(* IEC 61131-3 sources: BLM_BACKGROUND/src/PROGRAM_FILES/FB (part 3) *)

        _FB_Jog_Asse#STATE_JOG_ASSE_POS_ASSE_POSITIVE:
              IF (PosAsse.outputState<>GENERAL_STATE#STATE_END) THEN
                  PosAsse(AttesaResetAxes:=TRUE,
                                  axis:=Axes[Asse].PosAx,
                                  //direction:=BY_VALUE,
                                  //positioningMode:=pMode,
                                  position:=corsa,
                                  //velocityType:=DIRECT,
                                  velocity:=jogvel,
                                  //positiveAccelType:=DIRECT,
                                  //negativeAccelType:=DIRECT,
                                  positiveAccel:=jogacc,
                                  negativeAccel:=jogacc
                                  //velocityProfile:=TRAPEZOIDAL,
                                  //blendingMode:=INACTIVE,
                                  //mergeMode:=IMMEDIATELY,
                                  //nextCommand:=IMMEDIATELY
                                  );
              ELSE
                  PosAsse(AttesaResetAxes:=TRUE,
                                  axis:=Axes[Asse].PosAx,
                                  //direction:=BY_VALUE,
                                  //positioningMode:=pMode,
                                  position:=corsa,
                                  //velocityType:=DIRECT,
                                  velocity:=jogvel,
                                  //positiveAccelType:=DIRECT,
                                  //negativeAccelType:=DIRECT,
                                  positiveAccel:=jogacc,
                                  negativeAccel:=jogacc
                                  //velocityProfile:=TRAPEZOIDAL,
                                  //blendingMode:=INACTIVE,
                                  //mergeMode:=IMMEDIATELY,
                                  //nextCommand:=IMMEDIATELY
                                  );
                  CURRENT_STATE:=_FB_Jog_Asse#STATE_JOG_ASSE_JOG_PURO_NEGATIVO;
              END_IF;

        _FB_Jog_Asse#STATE_JOG_ASSE_JOG_PURO_NEGATIVO:
            //   {::ifdef BLOCCAGGIO_DX} %%%%% non c'e in config di machina
            //       IF Asse=W3 THEN
            //           AppoDirezione:=SN;
            //       ELSE
            //           AppoDirezione:=SN_SP;
            //       END_IF;
            //   {::else}
            //       AppoDirezione:=SN_SP;
            //   {::endif}
              IF ((r_minus.Q=TRUE) AND (Clk_plus=FALSE)) OR
                   ((Clk_plus=FALSE) AND (Clk_minus=TRUE) AND (r_rapid.Q=TRUE)) OR
                   ((Clk_minus=TRUE) AND (Clk_plus=FALSE) AND (f_rapid.q=TRUE)) THEN
                  IF OK_Condizione_Move_Asse(Asse:=Asse, Direzione:=AppoDirezione) THEN
                      reset_trace(Code:=TRC_SAFETY_JOG_DEVICES);
                      IF i_sys_varinc=0 THEN
                          // è in JOG puro e non incrementale
                          //limite negativo attivo
                          PosAx:= AsSynchronousAxisRef(Axes[asse].PosAx);
                          corsa:=PosAx^.PositionLimits_SW.MinPosition+EXTRALIMIT;
                          //corsa:=Axes[asse].PosAx.swlimit.minusposition+EXTRALIMIT;
                          pMode:=_EnumPositioningMode#ABSOLUTE;
                      ELSE
                          IF i_sys_varinc>=1 AND i_sys_varinc<=5 THEN
                              // valore fisso
                              corsa:=-INC[i_sys_varinc];

                              corsa:=INC_Enum#inc_0;
                              pMode:=_EnumPositioningMode#RELATIVE;
                            //   Axes[Asse].mcJogAxisInfo.Increment:=corsa; //???????
                            //   Axes[Asse].mcJogAxisInfo.ModeInc:=TRUE;
                          ELSE  // Quota target
                              //Se la quota supera il fine corsa la limita
                              PosAx:= AsSynchronousAxisRef(Axes[asse].PosAx);
                                IF pm[asse].MA_JOG_TARGET<PosAx^.PositionLimits_SW.MinPosition THEN
                                pm[asse].MA_JOG_TARGET:=PosAx^.PositionLimits_SW.MinPosition+EXTRALIMIT;
                              //IF pm[asse].MA_JOG_TARGET<Axes[asse].PosAx.swlimit.minusposition THEN
                                  //pm[asse].MA_JOG_TARGET:=Axes[asse].PosAx.swlimit.minusposition+EXTRALIMIT;
                              END_IF;
                              // se l^asse è oltre la quota target
                              PosAx:= AsSynchronousAxisRef(Axes[asse].PosAx);
                            //   IF Posax^.actualposition-Axes[Asse].Posax.servosettings.additionalcommandvalue[0]-0.1<pm[asse].MA_JOG_TARGET THEN ???
                            //       corsa:=PosAx^.PositionLimits_SW.MinPosition +EXTRALIMIT;
                            //   ELSE
                            //       // valore fisso
                            //       corsa:=pm[asse].MA_JOG_TARGET;
                            //   END_IF;
                              pMode:=_EnumPositioningMode#ABSOLUTE;
                          END_IF;
                      END_IF;
                  END_IF;
                  IF i_sys_monitoring<>0 OR i_sys_Accesslevel<=ACCESS_MANUTENTORE OR SbloccaMonitoring(Asse:=Asse)=TRUE THEN
                      IF Sbloccamonitoring(Asse:=Asse)=TRUE OR i_sys_monitoring=0 THEN
                          set_trace(Code:=TRC_MONITORING_DISABILITATO);
                      END_IF;// muove solo se in monitoring o con livello password alto e non è oltre il finecorsa negativo
                      PosAx:= AsSynchronousAxisRef(Axes[asse].PosAx);
                      IF Posax^.actualposition-0.01>PosAx^.PositionLimits_SW.MinPosition+EXTRALIMIT THEN
                          TestAsseUtensile(Asse);
                          i_sys_PosFinale[Asse]:=corsa;
                          IF (pMode=_EnumPositioningMode#RELATIVE AND USOPLCOpen) THEN
                              //Axes[Asse].mcJogAxisInfo.Enable:=TRUE;
                              Axes[Asse].MC_Axes.move_jog_param.JogBackward :=TRUE;
                              //Axes[Asse].mcJogAxisInfo.Backward:=TRUE;
                          ELSE
                              CURRENT_STATE:=_FB_Jog_Asse#STATE_JOG_ASSE_POS_ASSE_NEGATIVE;
                          END_IF;
                      ELSE
                          CURRENT_STATE:=_FB_Jog_Asse#STATE_JOG_ASSE_RILASCIO_PULSANTI;
                      END_IF;
                  ELSE
                      set_trace(Code:=TRC_JOG_NON_IN_MONITORING);
                      CURRENT_STATE:=_FB_Jog_Asse#STATE_JOG_ASSE_RILASCIO_PULSANTI;
                  END_IF;
              ELSE
                  CURRENT_STATE:=_FB_Jog_Asse#STATE_JOG_ASSE_RILASCIO_PULSANTI;
              END_IF;

        _FB_Jog_Asse#STATE_JOG_ASSE_POS_ASSE_NEGATIVE:
              IF (PosAsse.outputState<>GENERAL_STATE#STATE_END) THEN
                  PosAsse(AttesaResetAxes:=TRUE,
                                  axis:=Axes[Asse].PosAx,
                                  //direction:=BY_VALUE,
                                  positioningMode:=pMode,
                                  position:=corsa,
                                  //velocityType:=DIRECT,
                                  velocity:=jogvel,
                                  //positiveAccelType:=DIRECT,
                                  //negativeAccelType:=DIRECT,
                                  positiveAccel:=jogacc,
                                  negativeAccel:=jogacc
                                  //velocityProfile:=TRAPEZOIDAL,
                                  //blendingMode:=INACTIVE,
                                  //mergeMode:=IMMEDIATELY,
                                  //nextCommand:=IMMEDIATELY
                                  );
              ELSE
                  PosAsse(AttesaResetAxes:=TRUE,
                                  axis:=Axes[Asse].PosAx,
                                  //direction:=BY_VALUE,
                                  positioningMode:=pMode,
                                  position:=corsa,
                                  //velocityType:=DIRECT,
                                  velocity:=jogvel,
                                  //positiveAccelType:=DIRECT,
                                  //negativeAccelType:=DIRECT,
                                  positiveAccel:=jogacc,
                                  negativeAccel:=jogacc
                                  //velocityProfile:=TRAPEZOIDAL,
                                  //blendingMode:=INACTIVE,
                                  //mergeMode:=IMMEDIATELY,
                                  //nextCommand:=IMMEDIATELY
                                  );
                  CURRENT_STATE:=_FB_Jog_Asse#STATE_JOG_ASSE_RILASCIO_PULSANTI;
              END_IF;

        _FB_Jog_Asse#STATE_JOG_ASSE_RILASCIO_PULSANTI:
              //RILASCIATO TASTO ^+^ oppure RILASCIATO TASTO ^-^
              IF (f_plus.q=TRUE) OR (f_minus.q=TRUE) OR
                   ((r_plus.q=TRUE) AND (Clk_minus=TRUE)) OR
                   ((r_minus.q=TRUE) AND (Clk_plus=TRUE)) THEN
                  i_sys_posfinale[asse]:=-MY_BIG_VALUE_REAL;
                  IF (Axes[Asse].MC_Axes.State_move_jog.Busy) THEN
                    Axes[Asse].MC_Axes.move_jog_param.JogBackward :=FALSE;
                    Axes[Asse].MC_Axes.move_jog_param.JogForward :=FALSE;
                    //   Axes[Asse].mcJogAxisInfo.Backward:=FALSE;
                    //   Axes[Asse].mcJogAxisInfo.Forward:=FALSE;
                      //Axes[Asse].mcJogAxisInfo.Enable:=FALSE;
                  ELSE
                      StopAxis(asse:=asse  , Acceleration:=jogacc (*Deceleration:=jogacc*));
                  END_IF;
                  reset_trace(TRC_JOG_NON_IN_MONITORING);
                  reset_trace(Code:=TRC_MONITORING_DISABILITATO);
                  CURRENT_STATE:=GENERAL_STATE#STATE_END;
              ELSE
                  CURRENT_STATE:=GENERAL_STATE#STATE_END;
              END_IF;

          GENERAL_STATE#STATE_END:
              CURRENT_STATE:=GENERAL_STATE#STATE_INIT;

      END_CASE;
      OutputState:=CURRENT_STATE;
  END_FUNCTION_BLOCK

  FUNCTION_BLOCK FB_MuoviDispositivo

    VAR_EXTERNAL CONSTANT
        FIRST_DEVICE                          :INT;
    END_VAR

    VAR_INPUT
      Dispositivo    :INT;
      Stato          :INT;
    END_VAR
    VAR
      Esito            :BOOL;
      AppoStato        :INT;
      dret         		 :DINT;

          CURRENT_STATE				:INT:=GENERAL_STATE#STATE_INIT;
        //   {#ifndef ORBITALE}
        //       PinzaCoccodrillo	:FB_PinzaCoccodrillo;
        //   {#endif};
    END_VAR
      VAR_OUTPUT
          OutputState					:INT;
      END_VAR
      CASE CURRENT_STATE OF
          GENERAL_STATE#STATE_INIT:
              IF Dispositivo>=FIRST_DEVICE AND Dispositivo<=FIRST_DEVICE+_MAXDEVICES#MAXDEVICES-1 THEN
                //   {#ifdef ORBITALE}
                //       IF Disp[Dispositivo].TipoOut=DISP_OUT_V_C THEN
                //           AppoStato:=Stato;
                //           {#ifdef DH4010}
                //               IF Dispositivo=PINZA_SX OR Dispositivo=PINZA_DX THEN
                //                   //Gestione chiusura pinza su 2 posizioni. Se si parte da INTERMEDIO si può attivare LAVORO,
                //                   //altrimenti si attiva INTERMEDIO
                //                   IF Stato=LAVORO OR Stato=INTERMEDIO_PINZA THEN
                //                       IF Disp[Dispositivo].stato=INTERMEDIO_PINZA THEN
                //                           AppoStato:=LAVORO;
                //                       ELSE
                //                           AppoStato:=INTERMEDIO_PINZA;
                //                       END_IF;
                //                   END_IF;
                //                   IF Stato=RIPOSO OR Stato=INTERMEDIO_PINZA THEN
                //                       IF Disp[Dispositivo].stato=INTERMEDIO_PINZA THEN
                //                           AppoStato:=RIPOSO;
                //                       ELSE
                //                           AppoStato:=INTERMEDIO_PINZA;
                //                       END_IF;
                //                   END_IF;
                //               END_IF;
                //           {#endif}	//Fine DH4010
                //           Set_Disp_Position(Ndisp:=Dispositivo, Value:=AppoStato, TimerRisparmio:=TRUE);
                //           CURRENT_STATE:=GENERAL_STATE#STATE_END;
                //       ELSE
                //           set_disp(Ndisp:=Dispositivo, Stato:=Stato, TimerRisparmio:=TRUE);
                //           CURRENT_STATE:=GENERAL_STATE#STATE_END;
                //       END_IF;
                //   {#else}  //Fine ORBITALE
                //       IF Dispositivo=PINZA THEN
                //           IF cfg.UsoPinzaCoccoPneumatica=TRUE AND programmi[PROGRAMMA_JOG].PinzaCoccodrillo3Posizioni=TRUE THEN
                //               IF Stato=RIPOSO AND  Disp[PINZA].position=LAVORO THEN
                //                   AppoStato:=PREAPERTO;
                //               ELSE
                //                   AppoStato:=Stato;
                //               END_IF;
                //               CURRENT_STATE:=STATE_MUOVI_DISPOSITIVO_PINZA_COCCODRILLO;
                //           ELSE
                //               WriteDigitalOutput(NumOutput:=OUT_PREAPERTURA_PINZA_COCCODRILLO, Value:=FALSE);
                //               WriteDigitalOutput(NumOutput:=OUT_RESET_PINZA_COCCODRILLO_PREAPERTA, Value:=TRUE);
                //               set_disp(Ndisp:=Dispositivo, Stato:=Stato, TimerRisparmio:=TRUE);
                //               CURRENT_STATE:=GENERAL_STATE#STATE_END;
                //           END_IF;
                //       ELSE
                //           set_disp(Ndisp:=Dispositivo, Stato:=Stato, TimerRisparmio:=TRUE);
                //           CURRENT_STATE:=GENERAL_STATE#STATE_END;
                //       END_IF;
                //   {#endif}  //Fine NO ORBITALE
            //   ELSE
                  CURRENT_STATE:=GENERAL_STATE#STATE_END;
              END_IF;

        //   STATE_MUOVI_DISPOSITIVO_PINZA_COCCODRILLO:
        //   ;
            //   {#ifndef ORBITALE} %%%%
            //       IF PinzaCoccodrillo.OutputState<>GENERAL_STATE#STATE_END THEN
            //           PinzaCoccodrillo(Stato:=AppoStato,
            //                                            FlagStopPoint:=FALSE,
            //                                            Impostazione:=TRUE,
            //                                            Attesa:=FALSE,
            //                                            Trace:=FALSE);
            //       ELSE
            //           Esito:=PinzaCoccodrillo.ReturnValue;
            //           PinzaCoccodrillo();
            //           Disp[PINZA].position:=AppoStato;
            //           Disp[PINZA].stato:=AppoStato;
            //           CURRENT_STATE:=GENERAL_STATE#STATE_END;
            //       END_IF;
            //   {#endif};

          GENERAL_STATE#STATE_END:
              CURRENT_STATE:=GENERAL_STATE#STATE_INIT;

      END_CASE;
      OutputState:=CURRENT_STATE;
  END_FUNCTION_BLOCK

  FUNCTION_BLOCK FB_PosizionaSostegno
    VAR_INPUT
      Posizione :LREAL;
      Attesa    :BOOL:=TRUE;
    END_VAR
    VAR
      dret      :DINT;
      PosS1     :LREAL;
      OffsetS1  :LREAL;
      Programma :DINT;

          CURRENT_STATE				:INT:=GENERAL_STATE#STATE_INIT;
        //   Wait_Disp_Position	:FB_Wait_Disp_Position; %%%%
        //   PosAxeNoWait				:FB_PosAxeNoWait;
        //   WaitAxe							:FB_WaitAxe;
          EnableAxisBLM				:FB_EnableAxisBLM;
    END_VAR
      VAR_OUTPUT
          OutputState					:INT;
      END_VAR
      ;
    //   CASE CURRENT_STATE OF %%%%
    //       GENERAL_STATE#STATE_INIT:
    //           {#ifndef ORBITALE}
    //               {#ifdef SOSTEGNO_ELETTRICO}
    //                   //Impostazione dell^indice del pezzo attivo, se non siamo in AUTO il pezzo
    //                   //attivo da dove prendere i dati è 1
    //                   IF i_sys_OPMODE=AUTOMODE THEN
    //                       Programma:=i_sys_current_prog;
    //                   ELSE
    //                       Programma:=PROGRAMMA_JOG;
    //                   END_IF;
    //                   IF Assi[S1].PosAx.positioningState.homed=YES AND pm[S1].ma_stato_index=2 THEN
    //                       IF Programmi[Programma].diametro_tubo_sezione=TONDO THEN
    //                           //Gestione tubo tondo, la posizione S1 è calcolata direttamente da VGP
    //                           OffsetS1:=BlmMxToolsOffPezzo[(S1)].PosChiuso-
    //                                               BlmMxToolsOffPezzo[(S1)].Offset;
    //                           IF ABS(Posizione-RIPOSO)<=pm[S1].ma_tolerance OR
    //                                ABS(Posizione-BlmMxToolsOffPezzo[(S1)].PosAperto)<=pm[S1].ma_tolerance THEN
    //                               //Posizione bassa sostegno non si applica l^offset
    //                               PosS1:=BlmMxToolsOffPezzo[(S1)].PosAperto;
    //                           ELSE
    //                               IF ABS(Posizione-LAVORO)<=pm[S1].ma_tolerance THEN
    //                                   PosS1:=BlmMxToolsOffPezzo[(S1)].offset;
    //                               ELSE
    //                                   PosS1:=Posizione-OffsetS1;
    //                               END_IF;
    //                           END_IF;
    //                       ELSE
    //                           //Tubi non tondi la posizione di S1 dipende dalla posizione di Z1
    //                           IF ABS(Posizione-RIPOSO)<=pm[S1].ma_tolerance OR
    //                                ABS(Posizione-BlmMxToolsOffPezzo[(S1)].PosAperto)<=pm[S1].ma_tolerance THEN
    //                               //Posizione bassa sostegno non si applica l^offset
    //                               PosS1:=BlmMxToolsOffPezzo[(S1)].PosAperto;
    //                           ELSE
    //                               //Richiesta posizione alta occorre calcolarla in funzione di Z1
    //                               PosS1:=CalcS1daZ1(PosZ1:=Assi[Z1].PosAx.positioningState.actualPosition+
    //                                                                                Programmi[Programma].OffsetZ1RicSaldatura,
    //                                                                   Programma:=Programma,
    //                                                                   Sezione:=Programmi[Programma].diametro_tubo_sezione);
    //                           END_IF;
    //                       END_IF;
    //                       IF Attesa=FALSE AND Assi[S1].PosAx.control<>ACTIVE  THEN
    //                           CURRENT_STATE:=STATE_POSIZIONA_SOSTEGNO_ENABLE_SOSTEGNO;
    //                       ELSE
    //                           CURRENT_STATE:=STATE_POSIZIONA_SOSTEGNO_POS_SOSTEGNO_ELETTRICO;
    //                       END_IF;
    //                   ELSE
    //                       CURRENT_STATE:=GENERAL_STATE#STATE_END;
    //                   END_IF;
    //               {#else}
    //                   Set_disp_Position(Ndisp:=SUPPORT_TIRANT, Value:=Posizione, TimerRisparmio:=TRUE);
    //                   IF Attesa=TRUE THEN
    //                       CURRENT_STATE:=STATE_POSIZIONA_SOSTEGNO_WAIT_SOSTEGNO_PNEUMATICO;
    //                   ELSE
    //                       CURRENT_STATE:=GENERAL_STATE#STATE_END;
    //                   END_IF;
    //               {#endif}
    //           {#else}
    //               CURRENT_STATE:=GENERAL_STATE#STATE_END;
    //           {#endif};

    //       STATE_POSIZIONA_SOSTEGNO_POS_SOSTEGNO_ELETTRICO:
    //           {#ifdef SOSTEGNO_ELETTRICO}
    //               IF (PosAxeNoWait.outputState<>GENERAL_STATE#STATE_END) THEN
    //                   PosAxeNoWait(Quota:=PosS1, Asse:=S1);
    //               ELSE
    //                   PosAxeNoWait(Quota:=PosS1, Asse:=S1);
    //                   IF Attesa THEN
    //                       CURRENT_STATE:=STATE_POSIZIONA_SOSTEGNO_WAIT_SOSTEGNO_ELETTRICO;
    //                   ELSE
    //                       CURRENT_STATE:=GENERAL_STATE#STATE_END;
    //                   END_IF;
    //               END_IF;
    //           {#endif};

    //       STATE_POSIZIONA_SOSTEGNO_WAIT_SOSTEGNO_ELETTRICO:
    //           {#ifdef SOSTEGNO_ELETTRICO}
    //               IF (WaitAxe.outputState<>GENERAL_STATE#STATE_END) THEN
    //                   WaitAxe(Quota:=PosS1, Asse:=S1);
    //               ELSE
    //                   WaitAxe(Quota:=PosS1, Asse:=S1);
    //                   CURRENT_STATE:=GENERAL_STATE#STATE_END;
    //               END_IF;
    //           {#endif};

    //       STATE_POSIZIONA_SOSTEGNO_ENABLE_SOSTEGNO:
    //           {#ifdef SOSTEGNO_ELETTRICO}
    //               IF (EnableAxisBLM.outputState<>GENERAL_STATE#STATE_END) THEN
    //                   EnableAxisBLM(Asse:=assi[S1].PosAx,
    //                                               NumeroAsse:=S1,
    //                                               ModoAttesa:=IMMEDIATELY);
    //               ELSE
    //                   EnableAxisBLM(Asse:=assi[S1].PosAx,
    //                                               NumeroAsse:=S1,
    //                                               ModoAttesa:=IMMEDIATELY);
    //                   CURRENT_STATE:=GENERAL_STATE#STATE_END;
    //               END_IF;
    //           {#endif};

    //       STATE_POSIZIONA_SOSTEGNO_WAIT_SOSTEGNO_PNEUMATICO:
    //           {#ifndef SOSTEGNO_ELETTRICO}
    //               IF (Wait_Disp_Position.outputState<>GENERAL_STATE#STATE_END) THEN
    //                   Wait_Disp_Position(Device:=SUPPORT_TIRANT, Position:=LREAL_TO_INT(Posizione));
    //               ELSE
    //                   CURRENT_STATE:=GENERAL_STATE#STATE_END;
    //               END_IF;
    //           {#endif};

    //       GENERAL_STATE#STATE_END:
    //           CURRENT_STATE:=GENERAL_STATE#STATE_INIT;

    //   END_CASE;
    //   OutputState:=CURRENT_STATE;
  END_FUNCTION_BLOCK

/****************************************************************************************
 * DISABLES AXES AND PERFORMS A PUSH_ERROR IF THE MESSAGE CODE TO BE DISPLAYED IS GIVEN *
 ****************************************************************************************/

FUNCTION_BLOCK FB_SpegneAssi

    VAR_EXTERNAL
        Axes                            :ARRAY[_FIRST_AXIS#FIRST_AXIS.._FIRST_AXIS#FIRST_AXIS+_CONST_VAR_DEF._MAXIS#MAXAXIS-1] OF ax;
        pm                              : ARRAY[_FIRST_AXIS#FIRST_AXIS.._FIRST_AXIS#FIRST_AXIS+_CONST_VAR_DEF._MAXIS#MAXAXIS-1] OF AxisParameters;
    END_VAR

    VAR_EXTERNAL CONSTANT
        INACTIVE_DEACTIVATABLE_AXIS         :SINT;
    END_VAR

    VAR_INPUT
      Messaggio  	:DINT;
      Arresto    	:BOOL;
    END_VAR
    VAR
      PosAx         :REF_TO TO_SynchronousAxis;
      i          	:INT;
      dret      	:DINT;

          CURRENT_STATE			:INT:=GENERAL_STATE#STATE_INIT;
          CURRENT_AXIS			:INT;
          DisableAssi				:FB_DisableAxes;
    END_VAR
      VAR_OUTPUT
          OutputState				:INT;
      END_VAR
      CASE CURRENT_STATE OF
          GENERAL_STATE#STATE_INIT:
              CURRENT_AXIS:=_FIRST_AXIS#FIRST_AXIS-1;
              IF Messaggio>0 THEN
                  IF Arresto=TRUE THEN
                      CURRENT_STATE:=GENERAL_STATE#STATE_END;
                      dret:=Push_error(code:=Messaggio, Arresto:=TRUE);
                  ELSE
                      CURRENT_STATE:=GENERAL_STATE#STATE_END;
                      dret:=Push_error(code:=Messaggio, Arresto:=FALSE);
                  END_IF;
              END_IF;
              IF CURRENT_STATE<>GENERAL_STATE#STATE_END THEN
                  CURRENT_STATE:=_FB_SpegneAssi#STATE_SPEGNE_ASSI_LOOP_ASSI;
              END_IF;

            _FB_SpegneAssi#STATE_SPEGNE_ASSI_LOOP_ASSI:
              CURRENT_AXIS:=CURRENT_AXIS+1;
              IF CURRENT_AXIS<_MAXIS#MAXAXIS THEN
                  IF pm[CURRENT_AXIS].ma_asse_abilitato=TRUE AND pm[CURRENT_AXIS].ma_asse_installato<>INACTIVE_DEACTIVATABLE_AXIS THEN
                    PosAx:= AsSynchronousAxisRef(Axes[CURRENT_AXIS].PosAx);
                    IF PosAx^.StatusWord.%X7 THEN
                    //IF Axes[CURRENT_AXIS].PosAx.motionstatedata.motionstate=STANDSTILL THEN
                          CURRENT_STATE:=_FB_SpegneAssi#STATE_SPEGNE_ASSI_DISABLE_AXIS;
                      END_IF;
                  END_IF;
              ELSE
                  CURRENT_STATE:=GENERAL_STATE#STATE_END;
              END_IF;

            _FB_SpegneAssi#STATE_SPEGNE_ASSI_DISABLE_AXIS:
              IF DisableAssi.OutputState<>GENERAL_STATE#STATE_END THEN
                  DisableAssi(Asse:=CURRENT_AXIS(* , Regolatore:=ACTIVE, ProssimoCmd:=IMMEDIATELY*));
              ELSE
                  DisableAssi(Asse:=CURRENT_AXIS(* , Regolatore:=ACTIVE, ProssimoCmd:=IMMEDIATELY*));
                  CURRENT_STATE:=_FB_SpegneAssi#STATE_SPEGNE_ASSI_LOOP_ASSI;
              END_IF;

          GENERAL_STATE#STATE_END:
              CURRENT_STATE:=GENERAL_STATE#STATE_INIT;

      END_CASE;
      OutputState:=CURRENT_STATE;
  END_FUNCTION_BLOCK

  FUNCTION SbloccaMonitoring:BOOL

    VAR_EXTERNAL CONSTANT
        ACCESS_SAT           	:SINT;
    END_VAR

    VAR_EXTERNAL
        PagTabCorrezione                        :BOOL;
        pm                                      : ARRAY[_FIRST_AXIS#FIRST_AXIS.._FIRST_AXIS#FIRST_AXIS+_CONST_VAR_DEF._MAXIS#MAXAXIS-1] OF AxisParameters;
        i_sys_ACCESSLEVEL                       : INT;
        i_sys_monitoring                        : INT;
        access                                  :Access_Level;
    END_VAR

    VAR_INPUT
      Asse  :INT;
    END_VAR
    SbloccaMonitoring:=FALSE;
    IF PagTabCorrezione=TRUE THEN
      SbloccaMonitoring:=TRUE;
    ELSE
      IF Asse>=_FIRST_AXIS#FIRST_AXIS AND Asse<=_FIRST_AXIS#FIRST_AXIS+_MAXIS#MAXAXIS-1 THEN
        IF pm[Asse].ma_AsseInVGP=FALSE THEN
          //Asse non presente in VGP, non può quindi indicarne i limiti software
          SbloccaMonitoring:=TRUE;
        END_IF;

      END_IF;
      IF SbloccaMonitoring=FALSE THEN
        IF TestAsseBloccaggio(Asse)=TRUE OR TestAsseSpallamento(Asse)=TRUE THEN
          //Per gli assi bloccaggio e spallamento lo sbloccaggio del monitoring
          //può avvenire a partire da password SAT

        {::ifdef MCP_1900}
          SbloccaMonitoring:=(i_sys_accesslevel<=ACCESS_SAT AND i_sys_monitoring=0) ;
        {::else};
            SbloccaMonitoring:=(i_sys_accesslevel<=ACCESS_SAT AND i_sys_monitoring=0)

                            OR ((NOT MCPI_FEED_STOP AND NOT MCPI_SPINDLE_STOP) AND (i_sys_accesslevel<=access.jog_in_monitoring));
        {::endif};

        ELSE
          SbloccaMonitoring:=(i_sys_accesslevel<=access.jog_libero AND i_sys_monitoring=0)
                               {::ifndef MCP_1900}
                              OR ((NOT MCPI_FEED_STOP AND NOT MCPI_SPINDLE_STOP) AND (i_sys_accesslevel<=access.jog_in_monitoring));
                               {::endif};
        END_IF;
      END_IF;
    END_IF;
  END_FUNCTION

  FUNCTION OK_Condizione_Move_Asse:BOOL

    VAR_EXTERNAL CONSTANT
            TRC_SAFETY_JOG_DEVICES               :INT;
            PROGRAMMA_JOG                      	        :SINT;
            TRC_MACCHINA_PEZZO_DXSX                     :INT;
            MAXTOOLSOFFPEZZO                            :INT;
            W3 : INT;
            X1 :INT;
            U4 :INT;
            Z1 :INT;
            Y1 :INT;
            V1 :INT;
            L1 :INT;
            ERR_SLITTA_MOBILE_NON_A_ZERO                :DINT;
            FIRST_DEVICE                                :INT;
            PALETTA                                     :INT;
            ERR_BRACCIO_SOTTO_90                        :DINT;
            MAXDIGITALINPUT                             :INT;
            ACCESS_MANUTENTORE   	                    :SINT;
            INP_AL5_TRASLATORE_INDIETRO                 :INT;
            ERR_L1_TRASLATORE                           :DINT;
            ERR_TASSELLO_BLOCCAGGIO_DXSX                :DINT;

    END_VAR

    VAR_EXTERNAL
        pm                              : ARRAY[_FIRST_AXIS#FIRST_AXIS.._FIRST_AXIS#FIRST_AXIS+_CONST_VAR_DEF._MAXIS#MAXAXIS-1] OF AxisParameters;
        Axes                            :ARRAY[_FIRST_AXIS#FIRST_AXIS.._FIRST_AXIS#FIRST_AXIS+_CONST_VAR_DEF._MAXIS#MAXAXIS-1] OF ax;
        Disp                            :ARRAY[(FIRST_DEVICE)..(FIRST_DEVICE+_MAXDEVICES#MAXDEVICES-1)] OF Device;
        i_sys_current_prog	            :INT;
        i_sys_OPMODE                    : INT;
        BlmMxToolsOffPezzo              :ARRAY[0..MAXTOOLSOFFPEZZO-1] OF RigaUtDispositivo;
        Clk_Minus	                    :BOOL;
        mcpi_minus                      : BOOL;
        mcpi_plus                       : BOOL;
        Clk_Plus                        :BOOL;
        IAddress                        : ARRAY [0..MAXDIGITALINPUT] OF Digital_Input;
        i_sys_ACCESSLEVEL               : INT;
    END_VAR

    VAR_INPUT
      Asse      :INT;
      Direzione :INT;
    END_VAR

    VAR
      PosAx     : REF_TO TO_SynchronousAxis;
      iret      :INT;
      W3_Aperto :LREAL;
      TipoAl    :SINT;
      Programma :INT;
      Esito     :BOOL;
    END_VAR

      IF Asse<_FIRST_AXIS#FIRST_AXIS OR Asse>_FIRST_AXIS#FIRST_AXIS+_MAXIS#MAXAXIS-1 THEN
          OK_Condizione_Move_Asse:=FALSE;
      ELSE
            PosAx:= AsSynchronousAxisRef(Axes[Asse].posax);
          IF posax^.StatusWord.%X2 THEN
              OK_Condizione_Move_Asse:=FALSE;
          ELSE
              IF i_sys_OpMode=PI_COMMANDS_CODE#AUTOMODE THEN
                  Programma:=I_SYS_Current_Prog;
              ELSE
                  Programma:=PROGRAMMA_JOG;
              END_IF;
              OK_Condizione_Move_Asse:=TRUE;
            //   {
            //   #ifdef EFLEX_DH4010 %%%%
            //   }
            //       {
            //       #ifdef EFLEX
            //       }
            //           CASE Asse OF
            //               X1:
            //                   IF i_sys_SenzaTubo=FALSE AND disp[RULLI_TRASCINAMENTO].position<>LAVORO THEN
            //                       OK_Condizione_Move_Asse:=FALSE;
            //                   END_IF;
            //                   IF ABS(Assi[W1].PosAx.positioningState.actualPosition)>0.1 THEN
            //                       //Taglio non a riposo
            //                       set_trace(Code:=TRC_SAFETY_JOG_DEVICES, Asse:=W1);
            //                   END_IF;
            //               Q1:
            //                   IF (disp[TESTINA_1].position<>LAVORO OR disp[TESTINA_2].position<>LAVORO) AND mcpi_spindle_stop=TRUE THEN
            //                       OK_Condizione_Move_Asse:=FALSE;
            //                       iret:=Push_error(Code:=ERR_TESTINE_NO_BASSE);
            //                   END_IF;
            //           END_CASE;
            //       {
            //       #endif  //Fine EFLEX
            //       }
            //       {
            //       #ifdef DH4010
            //       }
            //           CASE Asse OF
            //               X1,X2,X3,X6:
            //                   IF Asse=X6 AND i_sys_SenzaTubo=FALSE AND disp[RULLI_TRASCINAMENTO].position<>LAVORO THEN
            //                       OK_Condizione_Move_Asse:=FALSE;
            //                       Set_Disp(Ndisp:=RULLI_TRASCINAMENTO, Stato:=LAVORO, TimerRisparmio:=TRUE);
            //                   END_IF;
            //                   OK_Condizione_Move_Asse:=TestCondizione(Dispositivo:=BLOCCAGGIO_3D, Stato:=RIPOSO, StatoOld:=OK_Condizione_Move_Asse);
            //                   OK_Condizione_Move_Asse:=TestCondizione(Dispositivo:=BLOCCAGGIO_2D, Stato:=RIPOSO, StatoOld:=OK_Condizione_Move_Asse);
            //                   OK_Condizione_Move_Asse:=TestCondizione(Dispositivo:=PINZA_SX, Stato:=RIPOSO, StatoOld:=OK_Condizione_Move_Asse);
            //                   OK_Condizione_Move_Asse:=TestCondizione(Dispositivo:=PINZA_DX, Stato:=RIPOSO, StatoOld:=OK_Condizione_Move_Asse);
            //                   OK_Condizione_Move_Asse:=TestCondizione(Dispositivo:=TAGLIO_SX, Stato:=RIPOSO, StatoOld:=OK_Condizione_Move_Asse);
            //                   OK_Condizione_Move_Asse:=TestCondizione(Dispositivo:=TAGLIO_DX, Stato:=RIPOSO, StatoOld:=OK_Condizione_Move_Asse);
            //                   OK_Condizione_Move_Asse:=TestCondizione(Dispositivo:=SMUSSATORE_PINZA, Stato:=RIPOSO, StatoOld:=OK_Condizione_Move_Asse);
            //                   OK_Condizione_Move_Asse:=TestCondizione(Dispositivo:=SMUSSATORE_UTENSILE, Stato:=RIPOSO, StatoOld:=OK_Condizione_Move_Asse);
            //                   IF Asse=X1 THEN
            //                       IF TestCoerenzaDispositivo(Dispositivo:=SCOMPARSA_SUPPORTO1_SX)=TRUE THEN
            //                           OK_Condizione_Move_Asse:=TestCondizione(Dispositivo:=SCOMPARSA_SUPPORTO1_SX, Stato:=LAVORO, StatoOld:=OK_Condizione_Move_Asse);
            //                       ELSE
            //                           OK_Condizione_Move_Asse:=FALSE;
            //                           iret:=Push_error(Code:=ERR_CONFIGURAZIONE_SOSTEGNI_DH4010, Asse:=SCOMPARSA_SUPPORTO1_SX);
            //                       END_IF;
            //                       IF TestCoerenzaDispositivo(Dispositivo:=SCOMPARSA_SUPPORTO2_SX)=TRUE THEN
            //                           OK_Condizione_Move_Asse:=TestCondizione(Dispositivo:=SCOMPARSA_SUPPORTO2_SX, Stato:=LAVORO, StatoOld:=OK_Condizione_Move_Asse);
            //                       ELSE
            //                           OK_Condizione_Move_Asse:=FALSE;
            //                           iret:=Push_error(Code:=ERR_CONFIGURAZIONE_SOSTEGNI_DH4010, Asse:=SCOMPARSA_SUPPORTO2_SX);
            //                       END_IF;
            //                   END_IF;
            //                   IF Asse=X2 OR Asse=X3 THEN
            //                       IF TestCoerenzaDispositivo(Dispositivo:=SCOMPARSA_SUPPORTO1_DX)=TRUE THEN
            //                           OK_Condizione_Move_Asse:=TestCondizione(Dispositivo:=SCOMPARSA_SUPPORTO1_DX, Stato:=LAVORO, StatoOld:=OK_Condizione_Move_Asse);
            //                       ELSE
            //                           OK_Condizione_Move_Asse:=FALSE;
            //                           iret:=Push_error(Code:=ERR_CONFIGURAZIONE_SOSTEGNI_DH4010, Asse:=SCOMPARSA_SUPPORTO1_DX);
            //                       END_IF;
            //                       IF TestCoerenzaDispositivo(Dispositivo:=SCOMPARSA_SUPPORTO2_DX)=TRUE THEN
            //                           OK_Condizione_Move_Asse:=TestCondizione(Dispositivo:=SCOMPARSA_SUPPORTO2_DX, Stato:=LAVORO, StatoOld:=OK_Condizione_Move_Asse);
            //                       ELSE
            //                           OK_Condizione_Move_Asse:=FALSE;
            //                           iret:=Push_error(Code:=ERR_CONFIGURAZIONE_SOSTEGNI_DH4010, Asse:=SCOMPARSA_SUPPORTO2_DX);
            //                       END_IF;
            //                   END_IF;
            //                   IF Asse=X6 THEN
            //                       IF TeAspoVersione2()=TRUE AND (r_plus.Q=TRUE OR r_minus.Q=TRUE) THEN
            //                           //Verifica solo sul fronte di salita dei tasti più o meno
            //                           OK_Condizione_Move_Asse:=NOT ReadDigitalInput(NumInput:=INP_ASPO_VER2_NON_PRONTO, Verifica:=TRUE) AND
            //                                                                            ReadDigitalInput(NumInput:=INP_ASPO_VER2_IN_AUTOMATICO, Verifica:=TRUE);
            //                       END_IF;
            //                   END_IF;
            //               Q1:
            //                   IF i_sys_monitoring=0 THEN
            //                       IF Assi[Y1].PosAx.positioningState.actualPosition>180 OR Assi[Y1].PosAx.positioningState.actualPosition<0 THEN
            //                           OK_Condizione_Move_Asse:=FALSE;
            //                           set_trace(Code:=TRC_JOG_NON_IN_MONITORING);
            //                       END_IF;
            //                   END_IF;
            //                   IF (disp[TESTINA_1_SX].position<>LAVORO OR disp[TESTINA_2_SX].position<>LAVORO) AND mcpi_spindle_stop=TRUE THEN
            //                       OK_Condizione_Move_Asse:=FALSE;
            //                       iret:=Push_error(Code:=ERR_TESTINE_NO_BASSE);
            //                   END_IF;
            //               Q2:
            //                   IF i_sys_monitoring=0 THEN
            //                       IF Assi[Y2].PosAx.positioningState.actualPosition>180 OR Assi[Y2].PosAx.positioningState.actualPosition<0 THEN
            //                           OK_Condizione_Move_Asse:=FALSE;
            //                           set_trace(Code:=TRC_JOG_NON_IN_MONITORING);
            //                       END_IF;
            //                   END_IF;
            //                   IF (disp[TESTINA_1_DX].position<>LAVORO OR disp[TESTINA_2_DX].position<>LAVORO) AND mcpi_spindle_stop=TRUE THEN
            //                       OK_Condizione_Move_Asse:=FALSE;
            //                       iret:=Push_error(Code:=ERR_TESTINE_NO_BASSE);
            //                   END_IF;
            //               Y1,Y2:
            //                   IF i_sys_monitoring=0 THEN
            //                       OK_Condizione_Move_Asse:=FALSE;
            //                       set_trace(Code:=TRC_JOG_NON_IN_MONITORING);
            //                   END_IF;
            //           END_CASE;
            //       {
            //       #endif  //Fine DH4010
            //       }
            //   {
            //   #else //Fine EFLEX_DH4010
            //   }
                  IF Utensili_DX_SX()=FALSE THEN
                      OK_Condizione_Move_Asse:=FALSE;
                      set_trace(Code:=TRC_MACCHINA_PEZZO_DXSX);
                  ELSE
                      IF ShadowMotorCheck()>=_FIRST_AXIS#FIRST_AXIS THEN
                          OK_Condizione_Move_Asse:=FALSE;
                      END_IF;
                  END_IF;
                  {::ifdef BLOCCAGGIO_DX}
                      //Impostazione quota di morsa destra aperta
                      W3_Aperto:=BlmMxToolsOffPezzo[(W3)].PosAperto-5;
                  {::endif}
                //   {
                //   #ifdef ORBITALE %%%%
                //   }
                //       {
                //       #ifdef RUNNER
                //       }
                //           CASE Asse OF
                //               {
                //               #ifdef FOUR_RUNNER_PLAUNO
                //               }
                //                   X1:
                //                       OK_Condizione_Move_Asse:=TestCondizione(Dispositivo:=PINZA_INTERNA, Stato:=RIPOSO, StatoOld:=OK_Condizione_Move_Asse);
                //                       {
                //                       #ifdef B1_B2
                //                       }
                //                           IF ABS(Assi[B1].PosAx.positioningState.actualPosition)>5 AND pm[B1].ma_asse_abilitato=TRUE THEN
                //                               OK_Condizione_Move_Asse:=FALSE;
                //                               set_trace(Code:=TRC_SAFETY_JOG_DEVICES, Asse:=FOUR_RIPC);
                //                           ELSE
                //                               IF ABS(Assi[B2].PosAx.positioningState.actualPosition)>5 AND pm[B2].ma_asse_abilitato=TRUE THEN
                //                                   OK_Condizione_Move_Asse:=FALSE;
                //                                   set_trace(Code:=TRC_SAFETY_JOG_DEVICES, Asse:=FOUR_RIPC);
                //                               END_IF;
                //                           END_IF;
                //                       {
                //                       #endif	//Fine B1_B2
                //                       }
                //                       {
                //                       #ifdef PLAUNO_PLAUNO_LIGHT
                //                       }
                //                           OK_Condizione_Move_Asse:=TestCondizione(Dispositivo:=BLOCCAGGIO_TUBO, Stato:=RIPOSO, StatoOld:=OK_Condizione_Move_Asse);
                //                       {
                //                       #endif	//Fine PLAUNO_PLAUNO_LIGHT
                //                       }
                //                       {
                //                       #ifdef IPC_DISPOSITIVO
                //                       }
                //                           OK_Condizione_Move_Asse:=TestCondizione(Dispositivo:=IPC_AVANZAMENTO, Stato:=RIPOSO, StatoOld:=OK_Condizione_Move_Asse);
                //                           IF cfg._4RUNNER_Mo1613=TRUE THEN
                //                               OK_Condizione_Move_Asse:=TestCondizione(Dispositivo:=IPC_LIGHT, Stato:=RIPOSO, StatoOld:=OK_Condizione_Move_Asse);
                //                           END_IF;
                //                       {
                //                       #endif	//Fine IPC_DISPOSITIVO
                //                       }
                //                       OK_Condizione_Move_Asse:=TestCondizione(Dispositivo:=PINZA_ACCOMPAG_CH_AP, Stato:=RIPOSO, StatoOld:=OK_Condizione_Move_Asse);
                //                       OK_Condizione_Move_Asse:=TestCondizione(Dispositivo:=FORATURA_MORSA, Stato:=RIPOSO, StatoOld:=OK_Condizione_Move_Asse);
                //                   V1, Q1:
                //                       OK_Condizione_Move_Asse:=TestCondizione(Dispositivo:=FORATURA_MORSA, Stato:=RIPOSO, StatoOld:=OK_Condizione_Move_Asse);
                //                       {
                //                       #ifdef FOUR_RUNNER
                //                       }
                //                           IF iaddress[INP_SBLOCCO_DX_SX].Port>-1 AND iaddress[INP_SBLOCCO_DX_SX].Bit>-1 THEN
                //                               IF Disp[BLOCCO_CANNOTTO].Position<>RIPOSO AND RunnerDXSX()=TRUE THEN
                //                                   Ok_condizione_move_Asse:=FALSE;
                //                                   Set_trace(Code:=TRC_SAFETY_JOG_DEVICES, Asse:=BLOCCO_CANNOTTO);
                //                               END_IF;
                //                           END_IF;
                //                       {
                //                       #endif //FINE FOUR_RUNNER
                //                       }
                //               {
                //               #endif	//Fine FOUR_RUNNER_PLAUNO
                //               }
                //               {
                //               #ifdef THREE_RUNNER
                //               }
                //                   X1:
                //                       OK_Condizione_Move_Asse:=TestCondizione(Dispositivo:=IPC_MORSA_STRAPPO, Stato:=RIPOSO, StatoOld:=OK_Condizione_Move_Asse);
                //                       OK_Condizione_Move_Asse:=TestCondizione(Dispositivo:=PINZA_INTERNA, Stato:=RIPOSO, StatoOld:=OK_Condizione_Move_Asse);
                //                       {
                //                       #ifdef B1_B2
                //                       }
                //                           IF ABS(Assi[B1].PosAx.positioningState.actualPosition)>5 THEN
                //                               OK_Condizione_Move_Asse:=FALSE;
                //                               set_trace(Code:=TRC_SAFETY_JOG_DEVICES, Asse:=THREE_RIPC);
                //                           ELSE
                //                               IF ABS(Assi[B2].PosAx.positioningState.actualPosition)>5 THEN
                //                                   OK_Condizione_Move_Asse:=FALSE;
                //                                   set_trace(Code:=TRC_SAFETY_JOG_DEVICES, Asse:=THREE_RIPC);
                //                               END_IF;
                //                           END_IF;
                //                       {
                //                       #endif	//Fine B1_B2
                //                       }
                //               {
                //               #endif	//Fine THREE_RUNNER
                //               }
                //           U1:
                //               IF Clk_plus=TRUE THEN
                //                   TestY1Safety();
                //               END_IF;
                //               {
                //               #ifndef PLAUNO_LIGHT
                //               }
                //                   IF (cfg._4RUNNER_4RForm_LevaScaricoScivolo) AND (disp[LEVA_SCARICO].Stato=LAVORO) THEN
                //                       Ok_Condizione_move_Asse:=FALSE;
                //                       iret:=Push_Error(Code:=ERR_MOVIMENTAZIONE_LEVA_SCARICO, Arresto:=TRUE);
                //                   END_IF;
                //               {
                //               #endif //FINE NO PLAUNO_LIGHT
                //               }
                //           W2:
                //               IF VerificaU2AllineataW1()=FALSE THEN
                //                   //Lo spintore per muoversi verso la morsa deve essere allineato, in caso contrario
                //                   //azzero il numero del dispositivo per fermarlo
                //                   OK_Condizione_Move_Asse:=FALSE;
                //                   set_trace(Code:=TRC_SAFETY_JOG_DEVICES, Asse:=U2);
                //               END_IF;
                //           U2:
                //               IF ABS(Assi[W2].PosAx.positioningState.actualPosition-pm[W2].Ma_Pos_Limit_Plus)>pm[W2].ma_tolerance THEN
                //                   //Spintore non indietro, non si può muovere U2
                //                   OK_Condizione_Move_Asse:=FALSE;
                //                   set_trace(Code:=trc_SICUREZZA_JOG_DISPOSITIVI, Asse:=W2);
                //               END_IF;
                //               IF Clk_plus=TRUE THEN
                //                   TestY1Safety();
                //               END_IF;
                //               {
                //               #ifdef A1_A2
                //               }
                //                   IF TestBloccaggio4RCPresente()=TRUE AND Disp[BLOCCAGGIO_4RC].Position<>RIPOSO THEN
                //                       OK_Condizione_Move_Asse:=FALSE;
                //                       set_trace(Code:=trc_SICUREZZA_JOG_DISPOSITIVI, Asse:=BLOCCAGGIO_4RC);
                //                   END_IF;
                //               {
                //               #endif	//Fine A1_A2
                //               }
                //               {
                //               #ifndef PLAUNO_LIGHT
                //               }
                //                   IF (cfg._4RUNNER_4RForm_LevaScaricoScivolo) AND (disp[LEVA_SCARICO].Stato=RIPOSO) THEN
                //                       OK_Condizione_Move_Asse:=FALSE;
                //                       iret:=Push_Error(Code:=ERR_MOVIMENTAZIONE_LEVA_SCARICO, Arresto:=TRUE);
                //                   END_IF;
                //               {
                //               #endif //FINE NO PLAUNO_LIGHT
                //               }
                //           END_CASE;
                //       {
                //       #endif	//Fine RUNNER
                //       }
                //   {
                //   #else	//Fine ORBITALE
                //   }
                      CASE Asse OF
                          X1:
                            //   {
                            //   #ifdef SMART %%%%
                            //   }
                            //       IF Disp[PALETTA].enable=TRUE AND Disp[PALETTA].stato<>LAVORO AND TestBasculanteCarico()=FALSE THEN
                            //           //Alzo paletta se basculante non è in posizione di carico
                            //           OK_Condizione_Move_Asse:=FALSE;
                            //           IF i_sys_OPMODE=MDAMODE THEN
                            //               set_trace(Code:=TRC_SAFETY_JOG_DEVICES, Asse:=PALETTA);
                            //           END_IF;
                            //       END_IF;
                            //   {
                            //   #else  //Fine SMART
                            //   }
                            //       IF Disp[PALETTA].stato<>LAVORO AND Disp[PALETTA].enable THEN
                            //           OK_Condizione_Move_Asse:=FALSE;
                            //           IF i_sys_OPMODE=MDAMODE THEN
                            //               set_trace(Code:=TRC_SAFETY_JOG_DEVICES, Asse:=PALETTA);
                            //           END_IF;
                            //       END_IF;
                            //   {
                            //   #endif  //Fine NO SMART
                            //   }
                            //   {
                            //   #ifdef SOSTEGNO_ELETTRICO
                            //   }
                            //       IF Assi[S1].PosAx.control<>ACTIVE THEN
                            //           OK_Condizione_Move_Asse:=FALSE;
                            //           EnableAxisBlm(Asse:=assi[S1].PosAx, NumeroAsse:=S1, ModoAttesa:=IMMEDIATELY);
                            //       ELSE
                            //           IF (Assi[S1].PosAx.positioningState.homed<>YES OR pm[S1].ma_stato_index<>2) AND
                            //                Assi[X1].PosAx.motionstatedata.commandvelocity<-1 THEN
                            //               OK_Condizione_Move_Asse:=FALSE;
                            //               iret:=Push_error(Code:=ERR_AXES_NO_INDEX);
                            //           END_IF;
                            //       END_IF;
                            //   {
                            //   #endif  //Fine SOSTEGNO_ELETTRICO
                            //   }
                            //   {
                            //   #ifdef MS0017
                            //   }
                            //       IF IndicaTipoAl()=TIPO_MS0017 AND mcpi_minus=TRUE THEN
                            //           //Non si può muovere in SN l^asse X1 se L1 è dentro gli ingombri della macchina
                            //           //tranne se l^operatore non esegue lo sblocca monitoring ed ha almeno la password manutentore
                            //           IF MCPI_FEED_STOP=TRUE OR MCPI_SPINDLE_STOP=TRUE OR i_sys_accesslevel>=ACCESS_PROGRAMMATORE THEN
                            //               IF Assi[L1].PosAx.PositioningState.ActualPosition>Programmi[Programma].DatiAL.MS0017_PosL1FuoriIng THEN
                            //                   IF TestRobotDaAl(Programma:=PROGRAMMA_JOG)=FALSE THEN
                            //                       OK_Condizione_Move_Asse:=FALSE;
                            //                       set_trace(Code:=TRC_SAFETY_JOG_DEVICES, Asse:=L1);
                            //                   END_IF;
                            //               END_IF;
                            //           END_IF;
                            //       END_IF;
                            //   {
                            //   #endif	//Fine MS0017
                            //   }
                        //   Y1:
                        //       //Non torna con la Y se è fuori la slitta mobile
                        //       {
                        //       #ifdef SMART_SMART_A
                        //       }
                        //           IF Assi[U4].posax.typeofaxis<>VIRTUAL_AXIS THEN
                        //               IF Assi[W4].PosAx.positioningState.actualPosition>0 THEN
                        //                   //Spallamento sul lato DX
                        //                   IF Clk_minus=TRUE AND Assi[U4].PosAx.positioningState.actualPosition>pm[U4].ma_standstill_pos_tol THEN
                        //                       OK_Condizione_Move_Asse:=FALSE;
                        //                       iret:=Push_error(Code:=ERR_SLITTA_MOBILE_NON_A_ZERO);
                        //                   END_IF;
                        //               ELSE
                        //                   //Spallamento sul lato SX
                        //                   IF Clk_plus=TRUE AND Assi[U4].PosAx.positioningState.actualPosition>pm[U4].ma_standstill_pos_tol THEN
                        //                       OK_Condizione_Move_Asse:=FALSE;
                        //                       iret:=Push_error(Code:=ERR_SLITTA_MOBILE_NON_A_ZERO);
                        //                   END_IF;
                        //               END_IF;
                        //           END_IF;
                        //       {
                        //       #else	//Fine SMART_SMART_A %%%%
                        //       }
                                //   {
                                //   #ifdef SLITTA_MOBILE_DX
                                //   }
                                        PosAx:=AsSynchronousAxisRef(Axes[U4].posax);
                                      IF posax^.VirtualAxis.Mode=UDINT#0 THEN
                                          IF Clk_minus=TRUE AND PosAx^.actualPosition>pm[U4].ma_standstill_pos_tol THEN
                                              OK_Condizione_Move_Asse:=FALSE;
                                              iret:=Push_error(Code:=ERR_SLITTA_MOBILE_NON_A_ZERO);
                                          END_IF;
                                      END_IF;
                            //       {
                            //       #endif	//Fine SLITTA_MOBILE_DX
                            //       }
                            //   {
                            //   #endif	//Fine NO SMART_SMART_A
                            //   }
                            //   {
                            //   #ifdef SLITTA_MOBILE_SX %%%%
                            //   }
                            //       //Non torna con la Y se è fuori la slitta mobile sinistra
                            //       IF Assi[U5].posax.typeofaxis<>VIRTUAL_AXIS THEN
                            //           IF Clk_minus=TRUE AND Assi[U5].PosAx.positioningState.actualPosition>pm[U5].ma_standstill_pos_tol THEN
                            //               OK_Condizione_Move_Asse:=FALSE;
                            //               iret:=Push_error(Code:=ERR_SLITTA_MOBILE_NON_A_ZERO);
                            //           END_IF;
                            //       END_IF;
                            //   {
                            //   #endif	//Fine SLITTA_MOBILE_SX
                            //   }
                            //   {
                            //   #ifdef MATRICE_ELETTRICA
                            //   }
                            //       IF TestAsseY2()=TRUE THEN
                            //           IF Clk_minus=TRUE OR Clk_plus=TRUE THEN
                            //               IF Assi[W3].PosAx.positioningState.actualPosition<W3_Aperto AND SbloccaMonitoring(Asse:=Y1)=FALSE THEN
                            //                   OK_Condizione_Move_Asse:=FALSE;
                            //                   set_trace(Code:=TRC_APRIRE_BLOCCAGGIO);
                            //               ELSE
                            //                   reset_trace(TRC_APRIRE_BLOCCAGGIO);
                            //               END_IF;
                            //           ELSE
                            //               reset_trace(TRC_APRIRE_BLOCCAGGIO);
                            //           END_IF;
                            //       END_IF;
                            //   {
                            //   #endif  //Fine MATRICE_ELETTRICA
                            //   }
                            //   {
                            //   #ifdef SMART
                            //   }
                            //       //Per la SMART occorre verificare la posizione della scomparsa rulli e del tassello
                            //       //bloccaggio DX/SX
                            //       IF cfg.tiposlittamobile=TIPO_SLITTA_ELETTRICA THEN
                            //           IF Assi[U4].PosAx.positioningState.actualPosition>U4_Scomparsa+0.2 THEN
                            //               IF Disp[BLOCCAGGIO_DXSX].enable AND cfg.bloccoscomparsabloccaggio=-1 THEN
                            //                   //Rulli in posizione diversa da scomparsa
                            //                   IF Clk_plus AND
                            //                        Assi[Y1].PosAx.positioningState.actualPosition>POSY_SCOMPBLOCC_SX AND
                            //                        Disp[BLOCCAGGIO_DXSX].Position<>LAVORO AND
                            //                        Assi[W4].PosAx.positioningState.actualPosition<0 THEN
                            //                       OK_Condizione_Move_Asse:=FALSE;
                            //                       iret:=Push_error(Code:=ERR_TASSELLO_BLOCCAGGIO_DXSX);
                            //                   ELSE
                            //                       IF Clk_minus AND
                            //                            Assi[Y1].PosAx.positioningState.actualPosition<POSY_SCOMPBLOCC_DX AND
                            //                            Disp[BLOCCAGGIO_DXSX].Position<>RIPOSO AND
                            //                            Assi[W4].PosAx.positioningState.actualPosition>0 THEN
                            //                           OK_Condizione_Move_Asse:=FALSE;
                            //                           iret:=Push_error(Code:=ERR_TASSELLO_BLOCCAGGIO_DXSX);
                            //                       END_IF;
                            //                   END_IF;
                            //               END_IF;
                            //           END_IF;
                            //       ELSE
                            //           IF Disp[DISAPPEARANCE_ROLLERS].enable=TRUE THEN
                            //               IF Disp[DISAPPEARANCE_ROLLERS].stato<>LAVORO THEN
                            //                   IF Disp[BLOCCAGGIO_DXSX].enable=TRUE AND cfg.bloccoscomparsabloccaggio=-1 THEN
                            //                       //Rulli in posizione diversa da scomparsa
                            //                       IF Clk_plus AND
                            //                            Assi[Y1].PosAx.positioningState.actualPosition>POSY_SCOMPBLOCC_SX AND
                            //                            Disp[BLOCCAGGIO_DXSX].Position<>LAVORO AND
                            //                            Assi[W4].PosAx.positioningState.actualPosition<0 THEN
                            //                           OK_Condizione_Move_Asse:=FALSE;
                            //                           iret:=Push_error(Code:=ERR_TASSELLO_BLOCCAGGIO_DXSX);
                            //                       ELSE
                            //                           IF Clk_minus AND
                            //                                Assi[Y1].PosAx.positioningState.actualPosition<POSY_SCOMPBLOCC_DX AND
                            //                                Disp[BLOCCAGGIO_DXSX].Position<>RIPOSO AND
                            //                                Assi[W4].PosAx.positioningState.actualPosition>0 THEN
                            //                               OK_Condizione_Move_Asse:=FALSE;
                            //                               iret:=Push_error(Code:=ERR_TASSELLO_BLOCCAGGIO_DXSX);
                            //                           END_IF;
                            //                       END_IF;
                            //                   END_IF;
                            //               END_IF;
                            //           ELSE
                            //               //Scomparsa rulli disabilitatata
                            //               IF Disp[BLOCCAGGIO_DXSX].enable=TRUE AND cfg.bloccoscomparsabloccaggio=-1 THEN
                            //                   IF Clk_plus AND
                            //                        Assi[Y1].PosAx.positioningState.actualPosition>POSY_SCOMPBLOCC_SX AND
                            //                        Disp[BLOCCAGGIO_DXSX].Position<>LAVORO AND
                            //                        Assi[W4].PosAx.positioningState.actualPosition<0 THEN
                            //                       OK_Condizione_Move_Asse:=FALSE;
                            //                       iret:=Push_error(Code:=ERR_TASSELLO_BLOCCAGGIO_DXSX);
                            //                   ELSE
                            //                       IF Clk_minus AND
                            //                            Assi[Y1].PosAx.positioningState.actualPosition<POSY_SCOMPBLOCC_DX AND
                            //                            Disp[BLOCCAGGIO_DXSX].Position<>RIPOSO AND
                            //                            Assi[W4].PosAx.positioningState.actualPosition>0 THEN
                            //                           OK_Condizione_Move_Asse:=FALSE;
                            //                           iret:=Push_error(Code:=ERR_TASSELLO_BLOCCAGGIO_DXSX);
                            //                       END_IF;
                            //                   END_IF;
                            //               END_IF;
                            //           END_IF;
                            //       END_IF;
                            //   {
                            //   #endif  //Fine SMART
                            //   }
                            //   {
                            //   #ifdef SMART_A
                            //   }
                            //       //Per la SMART occorre verificare la posizione della scomparsa rulli e del tassello
                            //       //bloccaggio DX/SX
                            //       IF Assi[U4].PosAx.positioningState.actualPosition>U4_Scomparsa+0.2 THEN
                            //           IF Disp[BLOCCAGGIO_DXSX].enable AND cfg.bloccoscomparsabloccaggio=-1 THEN
                            //               //Rulli in posizione diversa da scomparsa
                            //               IF Clk_plus AND
                            //                    Assi[Y1].PosAx.positioningState.actualPosition>POSY_SCOMPBLOCC_SX AND
                            //                    Disp[BLOCCAGGIO_DXSX].Position<>LAVORO AND
                            //                    Assi[W4].PosAx.positioningState.actualPosition<0 THEN
                            //                   OK_Condizione_Move_Asse:=FALSE;
                            //                   iret:=Push_error(Code:=ERR_TASSELLO_BLOCCAGGIO_DXSX);
                            //               ELSE
                            //                   IF Clk_minus AND
                            //                        Assi[Y1].PosAx.positioningState.actualPosition<POSY_SCOMPBLOCC_DX AND
                            //                        Disp[BLOCCAGGIO_DXSX].Position<>RIPOSO AND
                            //                        Assi[W4].PosAx.positioningState.actualPosition>0 THEN
                            //                       OK_Condizione_Move_Asse:=FALSE;
                            //                       iret:=Push_error(Code:=ERR_TASSELLO_BLOCCAGGIO_DXSX);
                            //                   END_IF;
                            //               END_IF;
                            //           END_IF;
                            //       END_IF;
                            //   {
                            //   #endif  //Fine SMART_A
                            //   }
                            //   {
                            //   #ifdef AL_BLM
                            //   }
                            //       {
                            //       #ifndef MS0017
                            //       }
                            //           //In caso di AL5 l^asse Y1 non si deve muovere se l^asse
                            //           //L1 non si trova in sicurezza
                            //           TipoAl:=IndicaTipoAl();
                            //           IF TipoAl=TIPO_AL5 OR TipoAl=TIPO_AL5_BUNDLE OR TipoAl=TIPO_AL5_FUTABA OR
                            //                TipoAl=TIPO_AL5_ROLAND OR TipoAl=TIPO_AL5_ROLAND_BUNDLE OR
                            //                TipoAl=TIPO_AL5_LUNGO OR TipoAl=TIPO_AL5_LUNGO_BUNDLE THEN
                            //               IF TestAl5Traslatore()=TRUE THEN
                            //                   IF IAddress[INP_AL5_TRASLATORE_INDIETRO].stato<>TRUE THEN
                            //                       iret:=Push_error(Code:=ERR_L1_TRASLATORE);
                            //                   END_IF;
                            //               ELSE
                            //                   IF Assi[L1].PosAx.PositioningState.ActualPosition>Programmi[PROGRAMMA_JOG].DatiAL.L1PosPrePresaTubo+pm[L1].MA_standstill_pos_tol THEN
                            //                       iret:=Push_error(Code:=ERR_L1_Y1);
                            //                   END_IF;
                            //               END_IF;
                            //           END_IF;
                            //       {
                            //       #endif  //Fine No MS0017
                            //       }
                            //   {
                            //   #endif  //Fine AL_BLM
                            //   }
                            //   ;
                          Z1:
                              IF Disp[PALETTA].stato<>DEVICES_STATUS#LAVORO AND Disp[PALETTA].enable THEN
                                  OK_Condizione_Move_Asse:=FALSE;
                                  IF i_sys_OPMODE=PI_COMMANDS_CODE#MDAMODE THEN
                                      set_trace(Code:=TRC_SAFETY_JOG_DEVICES, Axis:=PALETTA);
                                  END_IF;
                              END_IF;
                            //   {
                            //   #ifdef SOSTEGNO_ELETTRICO %%%%
                            //   }
                            //       IF Assi[S1].PosAx.control<>ACTIVE THEN
                            //           OK_Condizione_Move_Asse:=FALSE;
                            //           EnableAxisBlm(Asse:=assi[S1].PosAx, NumeroAsse:=S1, ModoAttesa:=IMMEDIATELY);
                            //       ELSE
                            //           IF (Assi[S1].PosAx.positioningState.homed<>YES OR pm[S1].ma_stato_index<>2) AND
                            //                Assi[X1].PosAx.motionstatedata.commandvelocity<-1 THEN
                            //               OK_Condizione_Move_Asse:=FALSE;
                            //               iret:=Push_error(Code:=ERR_AXES_NO_INDEX);
                            //           END_IF;
                            //       END_IF;
                            //   {
                            //   #endif  //Fine SOSTEGNO_ELETTRICO
                            //   }
                        //   Q1:
                            //   {
                            //   #ifdef AL_BLM
                            //   }
                            //       {
                            //       #ifndef MS0017
                            //       }
                            //           //In caso di AL5 l^asse Q1 per potersi muovere quando l^asse
                            //           //L1 non si trova in sicurezza, il braccio di curvatura deve essere
                            //           //a 0 o 180
                            //           TipoAl:=IndicaTipoAl();
                            //           IF TipoAl=TIPO_AL5 OR TipoAl=TIPO_AL5_BUNDLE OR TipoAl=TIPO_AL5_FUTABA OR
                            //                TipoAl=TIPO_AL5_ROLAND OR TipoAl=TIPO_AL5_ROLAND_BUNDLE OR
                            //                TipoAl=TIPO_AL5_LUNGO OR TipoAl=TIPO_AL5_LUNGO_BUNDLE THEN
                            //               IF TestAl5Traslatore()=TRUE THEN
                            //                   IF IAddress[INP_AL5_TRASLATORE_INDIETRO].stato<>TRUE AND
                            //                        i_sys_Accesslevel>ACCESS_MANUTENTORE THEN
                            //                       iret:=Push_error(Code:=ERR_L1_TRASLATORE);
                            //                   END_IF;
                            //               ELSE
                            //                   IF Assi[L1].PosAx.PositioningState.ActualPosition>Programmi[PROGRAMMA_JOG].DatiAL.L1PosPrePresaTubo+pm[L1].MA_standstill_pos_tol THEN
                            //                       IF Assi[Y1].PosAx.PositioningState.ActualPosition>1 AND
                            //                            Assi[Y1].PosAx.PositioningState.ActualPosition<179 THEN
                            //                           iret:=Push_error(Code:=ERR_L1_Y1_Q1);
                            //                       END_IF;
                            //                   END_IF;
                            //               END_IF;
                            //           END_IF;
                            //       {
                            //       #endif	//Fine No MS0017
                            //       }
                            //   {
                            //   #endif  //Fine AL_BLM
                            //   }
                            //   ;
                          V1:;
                            //   {
                            //   #ifndef MS0017
                            //   }
                            //       {
                            //       #ifdef AL_BLM
                            //       }
                            //           //In caso di AL5 l^asse V1 per potersi muovere quando l^asse
                            //           //L1 non si trova in sicurezza, il braccio di curvatura deve essere
                            //           //a 0 o 180
                            //           TipoAl:=IndicaTipoAl();
                            //           IF TipoAl=TIPO_AL5 OR TipoAl=TIPO_AL5_BUNDLE OR TipoAl=TIPO_AL5_FUTABA OR
                            //                TipoAl=TIPO_AL5_ROLAND OR TipoAl=TIPO_AL5_ROLAND_BUNDLE OR
                            //                TipoAl=TIPO_AL5_LUNGO OR TipoAl=TIPO_AL5_LUNGO_BUNDLE THEN
                            //               IF TestAl5Traslatore()=TRUE THEN
                            //                   IF IAddress[INP_AL5_TRASLATORE_INDIETRO].stato<>TRUE AND
                            //                        i_sys_Accesslevel>ACCESS_MANUTENTORE THEN
                            //                       iret:=Push_error(Code:=ERR_L1_TRASLATORE);
                            //                   END_IF;
                            //               ELSE
                            //                   IF Assi[L1].PosAx.PositioningState.ActualPosition>Programmi[PROGRAMMA_JOG].DatiAL.L1PosPrePresaTubo+pm[L1].MA_standstill_pos_tol THEN
                            //                       IF Assi[Y1].PosAx.PositioningState.ActualPosition>1 AND
                            //                            Assi[Y1].PosAx.PositioningState.ActualPosition<179 THEN
                            //                           iret:=Push_error(Code:=ERR_L1_Y1_R1);
                            //                       END_IF;
                            //                   END_IF;
                            //               END_IF;
                            //           END_IF;
                            //       {
                            //       #endif  //Fine AL_BLM
                            //       }
                            //   {
                            //   #endif  //Fine No MS0017
                            //   }
                            //   {
                            //   #ifdef BLOCCAGGIO_DX
                            //   }
                            //       {
                            //       #ifdef MATRICE_ELETTRICA
                            //       }
                            //           W3:
                            //               IF TestAsseY2()=TRUE THEN
                            //                   IF Direzione=SN THEN
                            //                       //In movimento in chiusura (SN) si deve verificare che la matrice sia nella stessa posizione del braccio
                            //                       //sia chiusa
                            //                       IF ABS(Assi[Y2].PosAx.positioningState.actualPosition-Assi[Y1].PosAx.positioningState.actualPosition)>pm[Y2].MA_standstill_pos_tol AND
                            //                            SbloccaMonitoring(Asse:=W3)=FALSE THEN
                            //                           IF Clk_minus=TRUE THEN
                            //                               set_trace(Code:=TRC_MATRICE_APERTA);
                            //                               OK_Condizione_Move_Asse:=FALSE;
                            //                           ELSE
                            //                               reset_trace(TRC_MATRICE_APERTA);
                            //                           END_IF;
                            //                       ELSE
                            //                           reset_trace(TRC_MATRICE_APERTA);
                            //                       END_IF;
                            //                   ELSE
                            //                       reset_trace(TRC_MATRICE_APERTA);
                            //                   END_IF;
                            //               END_IF;
                            //       {
                            //       #endif  //MATRICE_ELETTRICA
                            //       }
                            //       ;
                            //   {
                            //   #endif  //Fine BLOCCAGGIO_DX
                            //   }
                              {::ifdef SLITTA_MOBILE_DX}
                                //   U4:
                                //       {
                                //       #ifdef SMART_SMART_A %%%%
                                //       }
                                //           IF Assi[W4].PosAx.positioningState.actualPosition>0 THEN
                                //               IF Clk_plus=TRUE AND Assi[Y1].PosAx.positioningState.actualPosition<90 THEN
                                //                   OK_Condizione_Move_Asse:=FALSE;
                                //                   iret:=Push_error(Code:=ERR_BRACCIO_SOTTO_90);
                                //               END_IF;
                                //           ELSE
                                //               IF Clk_plus=TRUE AND Assi[Y1].PosAx.positioningState.actualPosition>90 THEN
                                //                   OK_Condizione_Move_Asse:=FALSE;
                                //                   iret:=Push_error(Code:=ERR_BRACCIO_SOTTO_90);
                                //               END_IF;
                                //           END_IF;
                                //       {
                                //       #else //Fine SMART_SMART_A
                                //       }
                                            PosAx:= AsSynchronousAxisRef(Axes[Y1].PosAx);
                                          IF Clk_plus=TRUE AND PosAx^.actualPosition<90 THEN
                                              OK_Condizione_Move_Asse:=FALSE;
                                              iret:=Push_error(Code:=ERR_BRACCIO_SOTTO_90);
                                          END_IF;
                            //           {
                            //           #endif  //Fine NO SMART_SMART_A
                            //           }
                             {::endif}
                            //   {
                            //   #ifdef SLITTA_MOBILE_SX
                            //   }
                            //       U5:
                            //           IF Clk_plus=TRUE AND Assi[Y1].PosAx.positioningState.actualPosition<90 THEN
                            //               OK_Condizione_Move_Asse:=FALSE;
                            //               iret:=Push_error(Code:=ERR_BRACCIO_SOTTO_90);
                            //           END_IF;
                            //   {
                            //   #endif  //Fine SLITTA_MOBILE_SX
                            //   }
                            //   {
                            //   #ifdef MATRICE_ELETTRICA
                            //   }
                            //       Y2:
                            //           IF TestAsseY2()=TRUE THEN
                            //               IF Clk_minus=TRUE OR Clk_plus=TRUE THEN
                            //                   IF Assi[W3].PosAx.positioningState.actualPosition<=W3_Aperto AND
                            //                        SbloccaMonitoring(Asse:=Y2)=FALSE THEN
                            //                       OK_Condizione_Move_Asse:=FALSE;
                            //                       set_trace(Code:=TRC_APRIRE_BLOCCAGGIO);
                            //                   ELSE
                            //                       reset_trace(TRC_APRIRE_BLOCCAGGIO);
                            //                   END_IF;
                            //               ELSE
                            //                   reset_trace(TRC_APRIRE_BLOCCAGGIO);
                            //               END_IF;
                            //           END_IF;
                            //   {
                            //   #endif  //Fine MATRICE_ELETTRICA
                            //   }
                            //   {
                            //   #ifdef SOSTEGNO_ELETTRICO
                            //   }
                            //       S1:
                            //           IF Assi[X1].PosAx.positioningState.actualPosition<MAX(i_sys_MAX_X_SOSTEGNO_ALTO, cfg.QuotaAbbassoSostegnoTirante)+pm[X1].ma_standstill_pos_tol THEN
                            //               OK_Condizione_Move_Asse:=FALSE;
                            //               set_trace(Code:=TRC_SAFETY_JOG_DEVICES, Asse:=X1);
                            //           END_IF;
                            //   {
                            //   #endif  //SOSTEGNO_ELETTRICO
                            //   }
                              {::ifdef AL_BLM}
                                  L1:
                                      IF TestAL5Traslatore()=TRUE THEN
                                          //Con traslatore orizzonatale tubo L1 può essere mosso solo con traslatore indietro
                                          IF IAddress[INP_AL5_TRASLATORE_INDIETRO].stato<>TRUE AND i_sys_Accesslevel>ACCESS_MANUTENTORE THEN
                                              OK_Condizione_Move_Asse:=FALSE;
                                              iret:=Push_error(Code:=ERR_L1_TRASLATORE);
                                          END_IF;
                                      END_IF;
                                    //   {
                                    //   #ifdef MS0017 %%%%
                                    //   }
                                    //       IF IndicaTipoAl()=TIPO_MS0017 AND mcpi_plus=TRUE THEN
                                    //           //Non si può muovere L1 in SP se X1 è inferiore alla quota di carico tranne se
                                    //           //l^operatore non esegue lo sblocca monitoring ed ha almeno la password manutentore
                                    //           IF MCPI_FEED_STOP=TRUE OR MCPI_SPINDLE_STOP=TRUE OR i_sys_accesslevel>=ACCESS_PROGRAMMATORE THEN
                                    //               IF Assi[X1].PosAx.PositioningState.ActualPosition<pm[X1].Ma_Pos_Limit_Plus_Attivo-EXTRALIMIT THEN
                                    //                   IF TestRobotDaAl(Programma:=PROGRAMMA_JOG)=FALSE THEN
                                    //                       OK_Condizione_Move_Asse:=FALSE;
                                    //                       set_trace(Code:=TRC_SAFETY_JOG_DEVICES, Asse:=X1);
                                    //                   END_IF;
                                    //               END_IF;
                                    //           END_IF;
                                    //       END_IF;
                                    //   {
                                    //   #endif  //Fine MS0017
                                    //   }
                              {::endif}
                            //   {
                            //   #ifdef BASCULANTE_ELETTRICO %%%%
                            //   }
                            //       B2:
                            //           IF BasculanteAvvio=FALSE THEN
                            //               IF Assi[V1].PosAx.positioningState.actualPosition-cfg.i_sys_postestabassaxmin>pm[V1].ma_standstill_pos_tol THEN
                            //                   iret:=Push_error(Code:=ERR_TESTA_NO_BASSA);
                            //                   OK_Condizione_Move_Asse:=FALSE;
                            //               END_IF;
                            //           END_IF;
                            //   {
                            //   #endif  //Fine BASCULANTE_ELETTRICO
                            //   }
                            //   {
                            //   #ifdef TAVOLI_ELETTRICI
                            //   }
                            //       //%%%%
                            //       T1:
                            //           IF Assi[Y1].PosAx.positioningState.actualPosition >= 90 AND Assi[Y1].PosAx.positioningState.actualPosition < 179 THEN
                            //               iret:=Push_error(Code:=ERR_BRACCIO_NON_OPPOSTO);
                            //               Ok_Condizione_Move_Asse:=FALSE;
                            //           END_IF;
                            //       T2:
                            //           IF Assi[Y1].PosAx.positioningState.actualPosition <= 90 AND Assi[Y1].PosAx.positioningState.actualPosition > 1 THEN
                            //               iret:=Push_error(Code:=ERR_BRACCIO_NON_OPPOSTO);
                            //               Ok_Condizione_Move_Asse:=FALSE;
                            //           END_IF;
                            //   {
                            //   #endif //FINE TAVOLI_ELETTRICI
                            //   }
                      END_CASE;
                //   {
                //   #endif  //Fine NO ORBITALE
                //   }
            //   {
            //   #endif  //Fine NO EFLEX_DH4010
            //   }
              IF (mcpi_minus=FALSE AND mcpi_plus=FALSE) OR OK_Condizione_Move_Asse=TRUE THEN
                  reset_trace(Code:=TRC_SAFETY_JOG_DEVICES);
              END_IF;
          END_IF;
    END_IF;
  END_FUNCTION

  //Verifica se la configurazione degli utensili inviata da VGP3D (per curvature DX/SX sullo stesso
//utensile è compatibile con la macchina attiva, oppure con un eventuale accessorio che
//consenta la curvatura DX/SX in processo
// {
// #ifndef EFLEX_DH4010 %%%%
// }
  FUNCTION Utensili_DX_SX:BOOL
    VAR
      i         			:INT;
      LatoUtensileDx  :INT;
      LatoUtensileSx  :INT;
    END_VAR
    ;
//     {
//     #ifdef CURVATURA
//     }
// 			LatoUtensileDx:=0;
// 			LatoUtensileSx:=0;
// 			Utensili_DX_SX:=FALSE;
// 			{
// 			#ifdef DXSX_PROCESSO
// 			}
// 				Utensili_DX_SX:=TRUE;
// 				GOTO Fine;
// 			{
// 			#endif	//Fine DXSX_PROCESSO
// 			}
// 			IF VerificaElectDXSX_PiegaInversa()=TRUE OR MO1094()=TRUE OR RunnerDXSX()=TRUE THEN
// 				Utensili_DX_SX:=TRUE;
// 			ELSE
// 				//E^ possibile effettuare la curvatura solo DX o solo SX
// 				FOR i:=1 TO MAXTOOLS DO
// 					IF BlmMxToolsDx[i].Qqt<>0 AND BlmMxToolsDx[i].Qtt<>0 THEN
// 						LatoUtensileDx:=DX;
// 					END_IF;
// 					IF BlmMxToolsSx[i].Qqt<>0 AND BlmMxToolsSx[i].Qtt<>0 THEN
// 						LatoUtensileSx:=SX;
// 					END_IF;
// 				END_FOR;
// 				IF LatoUtensileDx=DX AND LatoUtensileSx=SX THEN
// 					//Indicazione che è contemporanemante presente un utesile DXSX
// 					Utensili_DX_SX:=FALSE;
// 				ELSE
// 					//Presenti utensili o solo DX o solo SX, si verifica che siano
// 					//compatibili con il senso di curvatura della macchina
// 					IF (LatoUtensileDx=DX AND i_sys_senso_curvatura=DX) OR
// 						 (LatoUtensileSx=SX AND i_sys_senso_curvatura=SX) THEN
// 						Utensili_DX_SX:=TRUE;
// 					ELSE
// 						Utensili_DX_SX:=FALSE;
// 					END_IF;
// 				END_IF;
// 			END_IF;
// 			Fine:;
//     {
//     #else	//Fine CURVATURA
//     }
// 			Utensili_DX_SX:=TRUE;
//     {
//     #endif	//Fine CURVATURA
//     }
  END_FUNCTION
// {
// #endif	//Fine NO EFLEX_DH4010
// }

/*******************************************************************************
 * RETURNS TRUE IF THE TRANSLATOR CARRYING THE TUBE INTO THE MACHINE IS ACTIVE *
 *******************************************************************************/
FUNCTION TestAL5Traslatore:BOOL

    VAR_EXTERNAL
        OAddress                        : ARRAY [0..MAXDIGITALOUTPUT] OF Digital_Output;
        Disp                            :ARRAY[(FIRST_DEVICE)..(FIRST_DEVICE+_MAXDEVICES#MAXDEVICES-1)] OF Device;
    END_VAR

    VAR_EXTERNAL CONSTANT
        MAXDIGITALOUTPUT                    :INT;
        FIRST_DEVICE                        :INT;
        OUT_AL5_AVANTI_TRASLATORE           :INT;
        OUT_AL5_INDIETRO_TRASLATORE         :INT;
        AL5_TRASLATORE                      :INT;
    END_VAR

    {::ifdef AL_BLM}
      IF OAddress[OUT_AL5_AVANTI_TRASLATORE].port>-1 AND
         OAddress[OUT_AL5_AVANTI_TRASLATORE].bit>-1 AND
         OAddress[OUT_AL5_INDIETRO_TRASLATORE].port>-1 AND
         OAddress[OUT_AL5_INDIETRO_TRASLATORE].bit>-1 THEN
        TestAL5Traslatore:=TRUE;
        Disp[AL5_TRASLATORE].Enable:=TRUE;
      ELSE
        TestAL5Traslatore:=FALSE;
        Disp[AL5_TRASLATORE].Enable:=FALSE;
      END_IF;
    {::endif}
    ;
  END_FUNCTION

  FUNCTION OK_Condizione_Move_Dispositivo:BOOL

    VAR_EXTERNAL
        Disp                            :ARRAY[(FIRST_DEVICE)..(FIRST_DEVICE+_MAXDEVICES#MAXDEVICES-1)] OF Device;
        pm                              : ARRAY[_FIRST_AXIS#FIRST_AXIS.._FIRST_AXIS#FIRST_AXIS+_CONST_VAR_DEF._MAXIS#MAXAXIS-1] OF AxisParameters;
        Programmi                      :ARRAY[0.._CONST_VAR_DEF._MPROGRAMS#MAXPROGRAMS - UINT#1] OF Programma;
        Axes                            :ARRAY[_FIRST_AXIS#FIRST_AXIS.._FIRST_AXIS#FIRST_AXIS+_CONST_VAR_DEF._MAXIS#MAXAXIS-1] OF ax;
        cfg                             :_TYPE.Config_Struct;
        i_sys_MAX_X_SOSTEGNO_ALTO		:REAL;  //Quota massima X con sostegno alto, dopo si deve abbassare
        i_sys_monitoring                : INT ;
        Clk_Minus	                    :BOOL;
        Clk_Plus                        :BOOL;
    END_VAR

    VAR_EXTERNAL CONSTANT
        FIRST_DEVICE                          :INT;
        TRC_MACCHINA_PEZZO_DXSX               :INT;
        X1 : INT;
        Z1 : INT;
        W4 : INT;
        Y1 : INT;
        TRC_SAFETY_JOG_DEVICES              :INT;
        PROGRAM_JOG                      	:SINT;
        CLAMP                               :INT;  //32
        PALETTA                             :INT;  //33
        SUPPORT_TIRANT                      :INT;
        DISAPPEARANCE_ROLLERS               :INT;
        ERR_APRIRE_SLITTA_SPALLAMENTO       :DINT;
        LOCKING_DXSX                        :INT;
        POSY_SCOMPBLOCC_DX                	:REAL;
        POSY_SCOMPBLOCC_SX                	:REAL;
        ERR_TASSELLO_BLOCCAGGIO_DXSX        :DINT;
    END_VAR

    VAR_INPUT
      Dispositivo	:INT;
      Stato				:LREAL;
      TastoPiu		:BOOL;
      TastoMeno		:BOOL;
    END_VAR

    VAR
      PosAx             : REF_TO TO_SynchronousAxis;
      iret				:INT;
      dret				:DINT;
      i				    :INT;
      LimiteU2		    :REAL;
    END_VAR

      IF Dispositivo<FIRST_DEVICE OR Dispositivo>FIRST_DEVICE+_MAXDEVICES#MAXDEVICES-1 THEN
          OK_Condizione_Move_Dispositivo:=FALSE;
      ELSE
          OK_Condizione_Move_Dispositivo:=TRUE;
        //   {
        //   #ifdef EFLEX_DH4010 %%%%
        //   }
        //       {
        //       #ifdef DH4010
        //       }
        //           CASE Dispositivo OF
        //               SCOMP_PINZA_SX:
        //                   IF disp[PINZA_SX].stato<>RIPOSO THEN
        //                       OK_Condizione_Move_Dispositivo:=FALSE;
        //                   END_IF;
        //               SCOMP_PINZA_DX:
        //                   IF disp[PINZA_DX].stato<>RIPOSO THEN
        //                       OK_Condizione_Move_Dispositivo:=FALSE;
        //                   END_IF;
        //               SCOMP_MANIPOLATORE_3D:
        //                   IF Assi[X1].PosAx.PositioningState.ActualPosition+0.05<cfg.MinX1Manipolatore_Alto THEN
        //                       set_trace(Code:=TRC_SAFETY_JOG_DEVICES, Asse:=X1);
        //                       OK_Condizione_Move_Dispositivo:=FALSE;
        //                   ELSE
        //                       IF Assi[X2].PosAx.PositioningState.ActualPosition+0.05<cfg.MinX2Manipolatore_Alto THEN
        //                           set_trace(Code:=TRC_SAFETY_JOG_DEVICES, Asse:=X2);
        //                           OK_Condizione_Move_Dispositivo:=FALSE;
        //                       END_IF;
        //                   END_IF;
        //                   IF Disp[BLOCCAGGIO_3D].stato<>RIPOSO THEN
        //                       OK_Condizione_Move_Dispositivo:=FALSE;
        //                   END_IF;
        //                   IF ABS(Assi[Z1].PosAx.positioningState.actualPosition-65)>pm[Z1].ma_tolerance THEN
        //                       OK_Condizione_Move_Dispositivo:=FALSE;
        //                   END_IF;
        //                   IF Disp[BLOCCAGGIO_2D].Enable=TRUE AND TastoPiu=FALSE THEN
        //                       //Con il bloccaggio 2D abilitato non è possibile alzare il bloccaggio3D
        //                       set_trace(Code:=TRC_SAFETY_JOG_DEVICES, Asse:=BLOCCAGGIO_2D);
        //                       OK_Condizione_Move_Dispositivo:=FALSE;
        //                   END_IF;
        //               SCOMPARSA_SUPPORTO1_SX:
        //                   IF Disp[BLOCCAGGIO_SUPPORTO1_SX].Stato<>RIPOSO THEN
        //                       set_trace(Code:=TRC_SAFETY_JOG_DEVICES, Asse:=BLOCCAGGIO_SUPPORTO1_SX);
        //                       OK_Condizione_Move_Dispositivo:=FALSE;
        //                   END_IF;
        //                   IF Disp[SCOMPARSA_SUPPORTO1_SX].Limite2_Lavoro=Disp[SCOMPARSA_SUPPORTO1_SX].Limite2_Riposo THEN
        //                       OK_Condizione_Move_Dispositivo:=FALSE;
        //                       reset_trace(Code:=TRC_SAFETY_JOG_DEVICES);
        //                   END_IF;
        //               SCOMPARSA_SUPPORTO2_SX:
        //                   IF Disp[BLOCCAGGIO_SUPPORTO2_SX].Stato<>RIPOSO THEN
        //                       set_trace(Code:=TRC_SAFETY_JOG_DEVICES, Asse:=BLOCCAGGIO_SUPPORTO2_SX);
        //                       OK_Condizione_Move_Dispositivo:=FALSE;
        //                   END_IF;
        //                   IF Disp[SCOMPARSA_SUPPORTO2_SX].Limite2_Lavoro=Disp[SCOMPARSA_SUPPORTO2_SX].Limite2_Riposo THEN
        //                       OK_Condizione_Move_Dispositivo:=FALSE;
        //                       reset_trace(Code:=TRC_SAFETY_JOG_DEVICES);
        //                   END_IF;
        //               SCOMPARSA_SUPPORTO1_DX:
        //                   IF Disp[BLOCCAGGIO_SUPPORTO1_DX].Stato<>RIPOSO THEN
        //                       set_trace(Code:=TRC_SAFETY_JOG_DEVICES, Asse:=BLOCCAGGIO_SUPPORTO1_DX);
        //                       OK_Condizione_Move_Dispositivo:=FALSE;
        //                   END_IF;
        //                   IF Disp[SCOMPARSA_SUPPORTO1_DX].Limite2_Lavoro=Disp[SCOMPARSA_SUPPORTO1_DX].Limite2_Riposo THEN
        //                       OK_Condizione_Move_Dispositivo:=FALSE;
        //                       reset_trace(Code:=TRC_SAFETY_JOG_DEVICES);
        //                   END_IF;
        //               SCOMPARSA_SUPPORTO2_DX:
        //                   IF Disp[BLOCCAGGIO_SUPPORTO2_DX].Stato<>RIPOSO THEN
        //                       set_trace(Code:=TRC_SAFETY_JOG_DEVICES, Asse:=BLOCCAGGIO_SUPPORTO2_DX);
        //                       OK_Condizione_Move_Dispositivo:=FALSE;
        //                   END_IF;
        //                   IF Disp[SCOMPARSA_SUPPORTO2_DX].Limite2_Lavoro=Disp[SCOMPARSA_SUPPORTO2_DX].Limite2_Riposo THEN
        //                       OK_Condizione_Move_Dispositivo:=FALSE;
        //                       reset_trace(Code:=TRC_SAFETY_JOG_DEVICES);
        //                   END_IF;
        //               BLOCCAGGIO_SUPPORTO1_SX:
        //                   IF Disp[SCOMPARSA_SUPPORTO1_SX].Position<>Disp[SCOMPARSA_SUPPORTO1_SX].Limite_Riposo THEN
        //                       OK_Condizione_Move_Dispositivo:=FALSE;
        //                       set_trace(Code:=TRC_SAFETY_JOG_DEVICES, Asse:=BLOCCAGGIO_SUPPORTO1_SX);
        //                   END_IF;
        //               BLOCCAGGIO_SUPPORTO2_SX:
        //                   IF Disp[SCOMPARSA_SUPPORTO2_SX].Position<>Disp[SCOMPARSA_SUPPORTO2_SX].Limite_Riposo THEN
        //                       OK_Condizione_Move_Dispositivo:=FALSE;
        //                       set_trace(Code:=TRC_SAFETY_JOG_DEVICES, Asse:=BLOCCAGGIO_SUPPORTO2_SX);
        //                   END_IF;
        //               BLOCCAGGIO_SUPPORTO1_DX:
        //                   IF Disp[SCOMPARSA_SUPPORTO1_DX].Position<>Disp[SCOMPARSA_SUPPORTO1_DX].Limite_Riposo THEN
        //                       OK_Condizione_Move_Dispositivo:=FALSE;
        //                       set_trace(Code:=TRC_SAFETY_JOG_DEVICES, Asse:=BLOCCAGGIO_SUPPORTO1_DX);
        //                   END_IF;
        //               BLOCCAGGIO_SUPPORTO2_DX:
        //                   IF Disp[SCOMPARSA_SUPPORTO2_DX].Position<>Disp[SCOMPARSA_SUPPORTO2_DX].Limite_Riposo THEN
        //                       OK_Condizione_Move_Dispositivo:=FALSE;
        //                       set_trace(Code:=TRC_SAFETY_JOG_DEVICES, Asse:=BLOCCAGGIO_SUPPORTO2_DX);
        //                   END_IF;
        //               SCOMP1_SX, SCOMP2_SX:
        //                   IF readdigitalinput(NumInput:=INP_PALPATOIO_1_AVANTI_TESTA_SX)=TRUE AND Disp[PALPATORE_1_SX].Enable=TRUE THEN
        //                       OK_Condizione_Move_Dispositivo:=FALSE;
        //                       set_trace(Code:=TRC_PALPATORE_1_SX, Asse:=PALPATORE_1_SX);
        //                   ELSE
        //                       IF readdigitalinput(NumInput:=INP_PALPATOIO_2_AVANTI_TESTA_SX)=TRUE AND Disp[PALPATORE_2_SX].Enable=TRUE THEN
        //                           OK_Condizione_Move_Dispositivo:=FALSE;
        //                           set_trace(Code:=TRC_PALPATORE_2_SX, Asse:=PALPATORE_2_SX);
        //                       ELSE
        //                           IF readdigitalinput(NumInput:=INP_PALPATOIO_3_AVANTI_TESTA_SX)=TRUE AND Disp[PALPATORE_3_SX].Enable=TRUE THEN
        //                               OK_Condizione_Move_Dispositivo:=FALSE;
        //                               set_trace(Code:=TRC_PALPATORE_3_SX, Asse:=PALPATORE_3_SX);
        //                           ELSE
        //                               IF readdigitalinput(NumInput:=INP_PALPATOIO_4_AVANTI_TESTA_SX)=TRUE AND Disp[PALPATORE_4_SX].Enable=TRUE THEN
        //                                   OK_Condizione_Move_Dispositivo:=FALSE;
        //                                   set_trace(Code:=TRC_PALPATORE_4_SX, Asse:=PALPATORE_4_SX);
        //                               END_IF;
        //                           END_IF;
        //                       END_IF;
        //                   END_IF;
        //               SCOMP1_DX, SCOMP2_DX:
        //                   IF readdigitalinput(NumInput:=INP_PALPATOIO_1_AVANTI_TESTA_DX)=TRUE AND Disp[PALPATORE_1_DX].Enable=TRUE THEN
        //                       OK_Condizione_Move_Dispositivo:=FALSE;
        //                       set_trace(Code:=TRC_PALPATORE_1_DX, Asse:=PALPATORE_1_DX);
        //                   ELSE
        //                       IF readdigitalinput(NumInput:=INP_PALPATOIO_2_AVANTI_TESTA_DX)=TRUE AND Disp[PALPATORE_2_DX].Enable=TRUE THEN
        //                           OK_Condizione_Move_Dispositivo:=FALSE;
        //                           set_trace(Code:=TRC_PALPATORE_2_DX, Asse:=PALPATORE_2_DX);
        //                       ELSE
        //                           IF readdigitalinput(NumInput:=INP_PALPATOIO_3_AVANTI_TESTA_DX)=TRUE AND Disp[PALPATORE_3_DX].Enable=TRUE THEN
        //                               OK_Condizione_Move_Dispositivo:=FALSE;
        //                               set_trace(Code:=TRC_PALPATORE_3_DX, Asse:=PALPATORE_3_DX);
        //                           ELSE
        //                               IF readdigitalinput(NumInput:=INP_PALPATOIO_4_AVANTI_TESTA_DX)=TRUE AND Disp[PALPATORE_4_DX].Enable=TRUE THEN
        //                                   OK_Condizione_Move_Dispositivo:=FALSE;
        //                                   set_trace(Code:=TRC_PALPATORE_4_DX, Asse:=PALPATORE_4_DX);
        //                               END_IF;
        //                           END_IF;
        //                       END_IF;
        //                   END_IF;
        //           END_CASE;
        //       {
        //       #endif  //Fine DH4010
        //       }
        //   {
        //   #else  //Fine EFLEX_DH4010
        //   }
              IF Utensili_DX_SX()=FALSE THEN
                  set_trace(Code:=TRC_MACCHINA_PEZZO_DXSX);
                  OK_Condizione_Move_Dispositivo:=FALSE;
              ELSE
                  IF  ShadowMotorCheck()>=_FIRST_AXIS#FIRST_AXIS THEN
                      OK_Condizione_Move_Dispositivo:=FALSE;
                  END_IF;
              END_IF;
            //   {
            //   #ifdef PLAUNO_LIGHT %%%%
            //   }
            //       {
            //       #ifdef TAVOLI_SERPENTINE
            //       }
            //           CASE Dispositivo OF
            //               TAVOLO_POST_ORIZZONTALE, TAVOLO_POST_ORIZZ_DX, TAVOLO_POST_ORIZZ_SX, TAVOLO_POST_ROTAZIONE:
            //                   //Consentiti movimenti di chiusura tavoli verso la macchina solo con Z1 a 0° o 180°
            //                   IF Stato=RIPOSO THEN
            //                       IF ABS(Assi[Z1].PosAx.positioningState.actualPosition-0)>pm[Z1].ma_standstill_pos_tol AND
            //                            ABS(Assi[Z1].PosAx.positioningState.actualPosition-180)>pm[Z1].ma_standstill_pos_tol THEN
            //                           OK_Condizione_Move_Dispositivo:=FALSE;
            //                           set_trace(Code:=TRC_SAFETY_JOG_DEVICES, Asse:=Z1);
            //                       END_IF;
            //                   END_IF;
            //               TAVOLO_ANT_ORIZZONTALE:
            //                   IF Stato=RIPOSO THEN
            //                       //Consentiti movimenti di chiusura tavolo verso la macchina solo con Z1 a 0° o 180°
            //                       IF ABS(Assi[Z1].PosAx.positioningState.actualPosition-0)>pm[Z1].ma_standstill_pos_tol AND
            //                            ABS(Assi[Z1].PosAx.positioningState.actualPosition-180)>pm[Z1].ma_standstill_pos_tol THEN
            //                           OK_Condizione_Move_Dispositivo:=FALSE;
            //                           set_trace(Code:=TRC_SAFETY_JOG_DEVICES, Asse:=Z1);
            //                       END_IF;
            //                   END_IF;
            //                   IF Stato=LAVORO THEN
            //                       //Richiesta apertura tavolo orizzontale
            //                       IF ReadDigitalInput(NumInput:=INP_TAVOLO_ANTERIORE_ALTO, Verifica:=TRUE)=FALSE THEN
            //                           //Tavolo non è alto
            //                           IF RunnerDXSX()=TRUE THEN
            //                               IF Assi[Y1].PosAx.positioningState.actualPosition>1 AND Assi[Z1].PosAx.positioningState.actualPosition<179 THEN
            //                                   //Con DXSX in processo non si può muovere se l^asse Y1 non è a 0° o 180°
            //                                   OK_Condizione_Move_Dispositivo:=FALSE;
            //                                   set_trace(Code:=TRC_SAFETY_JOG_DEVICES, Asse:=Y1);
            //                               END_IF;
            //                           ELSE
            //                               IF Assi[Y1].PosAx.positioningState.actualPosition>1 THEN
            //                                   //Non si può muovere se l^asse Y1 non è a 0°
            //                                   OK_Condizione_Move_Dispositivo:=FALSE;
            //                                   set_trace(Code:=TRC_SAFETY_JOG_DEVICES, Asse:=Y1);
            //                               END_IF;
            //                           END_IF;
            //                       END_IF;
            //                   END_IF;
            //               TAVOLO_ANT_ROTAZIONE:
            //                   //Consentiti movimenti di chiusura tavoli verso la macchina solo con Z1 a 0° o 180°
            //                   IF Stato=RIPOSO THEN
            //                       IF ABS(Assi[Z1].PosAx.positioningState.actualPosition-0)>pm[Z1].ma_standstill_pos_tol AND
            //                           ABS(Assi[Z1].PosAx.positioningState.actualPosition-180)>pm[Z1].ma_standstill_pos_tol THEN
            //                           OK_Condizione_Move_Dispositivo:=FALSE;
            //                           set_trace(Code:=TRC_SAFETY_JOG_DEVICES, Asse:=Z1);
            //                       END_IF;
            //                   END_IF;
            //                   IF ReadDigitalInput(NumInput:=INP_TAVOLO_ANTERIORE_FUORI_INGOMBRO, Verifica:=TRUE)=TRUE THEN
            //                       //Tavolo anteriore orizzontale aperto
            //                       IF RunnerDXSX()=TRUE THEN
            //                           IF Assi[Y1].PosAx.positioningState.actualPosition>1 AND Assi[Z1].PosAx.positioningState.actualPosition<179 THEN
            //                               //Con DXSX in processo non si può muovere se l^asse Y1 non è a 0° o 180°
            //                               OK_Condizione_Move_Dispositivo:=FALSE;
            //                               set_trace(Code:=TRC_SAFETY_JOG_DEVICES, Asse:=Y1);
            //                           END_IF;
            //                       ELSE
            //                           IF Assi[Y1].PosAx.positioningState.actualPosition>1 THEN
            //                               //Non si può muovere se l^asse Y1 non è a 0°
            //                               OK_Condizione_Move_Dispositivo:=FALSE;
            //                               set_trace(Code:=TRC_SAFETY_JOG_DEVICES, Asse:=Y1);
            //                           END_IF;
            //                       END_IF;
            //                   END_IF;
            //           END_CASE;
            //       {
            //       #endif  //Fine TAVOLI_SERPENTINE
            //       }
            //   {
            //   #else	//Fine PLAUNO_LIGHT
            //   }
                  CASE Dispositivo OF
                    //   {
                    //   #ifdef RUNNER %%%%
                    //   }
                    //       LEVA_SCARICO:
                    //           IF cfg._4RUNNER_TipoTaglioEsterno=TAGLIO_4RTL THEN
                    //               LimiteU2:=cfg._4RUNNER_Pos_U2_LEVA_ALTA;
                    //           ELSE
                    //               LimiteU2:=cfg._4RUNNER_Pos_U2_LEVA_ALTA_4RC;
                    //           END_IF;
                    //           IF Assi[U2].PosAx.positioningState.actualPosition>LimiteU2 THEN
                    //               OK_Condizione_Move_Dispositivo:=FALSE;
                    //               set_trace(Code:=trc_SICUREZZA_JOG_DISPOSITIVI, Asse:=U2);
                    //           END_IF;
                    //           IF ((Assi[U1].PosAx.PositioningState.ActualPosition<=cfg._4RUNNER_U1PosTaglio) AND (Assi[U1].PosAx.PositioningState.ActualPosition>=pm[U1].ma_pos_limit_minus + 50)) AND (cfg._4RUNNER_4RForm_LevaScaricoScivolo) AND (Stato=LAVORO) THEN
                    //               OK_Condizione_Move_Dispositivo:=FALSE;
                    //               iret:=Push_Error(Code:=ERR_MOVIMENTAZIONE_LEVA_SCARICO, Arresto:=TRUE);
                    //           END_IF;
                    //           IF (Assi[U2].PosAx.PositioningState.ActualPosition>0) AND (cfg._4RUNNER_4RForm_LevaScaricoScivolo) AND (Stato=RIPOSO) THEN
                    //               OK_Condizione_Move_Dispositivo:=FALSE;
                    //               iret:=Push_Error(Code:=ERR_MOVIMENTAZIONE_LEVA_SCARICO, Arresto:=TRUE);
                    //           END_IF;
                    //           {
                    //           #ifdef THREE_RUNNER
                    //           }
                    //               IPC_STRAPPO:
                    //                   IF r_minus.Q=TRUE THEN
                    //                       IF Disp[IPC_MORSA_STRAPPO].stato<>RIPOSO THEN
                    //                           OK_Condizione_Move_Dispositivo:=FALSE;
                    //                           set_trace(Code:=TRC_SAFETY_JOG_DEVICES, Asse:=IPC_MORSA_STRAPPO);
                    //                       END_IF;
                    //                   END_IF;
                    //               IPC_STRAPPO_SCARICO:
                    //                   IF r_minus.Q=TRUE THEN
                    //                       IF Disp[IPC_MORSA_STRAPPO].stato<>RIPOSO THEN
                    //                           OK_Condizione_Move_Dispositivo:=FALSE;
                    //                           set_trace(Code:=TRC_SAFETY_JOG_DEVICES, Asse:=IPC_MORSA_STRAPPO);
                    //                       END_IF;
                    //                       IF Disp[IPC_STRAPPO].stato<>RIPOSO THEN
                    //                           OK_Condizione_Move_Dispositivo:=FALSE;
                    //                           set_trace(Code:=TRC_SAFETY_JOG_DEVICES, Asse:=IPC_STRAPPO);
                    //                       END_IF;
                    //                   END_IF;
                    //           {
                    //           #endif	//Fine THREE_RUNNER
                    //           }
                    //           {
                    //           #ifdef A1_A2
                    //           }
                    //               IF TestBloccaggio4RCPresente()=TRUE AND Disp[BLOCCAGGIO_4RC].Position<>RIPOSO THEN
                    //                   OK_Condizione_Move_Dispositivo:=FALSE;
                    //                   set_trace(Code:=trc_SICUREZZA_JOG_DISPOSITIVI, Asse:=BLOCCAGGIO_4RC);
                    //               END_IF;
                    //           {
                    //           #endif	//Fine A1_A2
                    //           }
                    //           {
                    //           #ifdef FOUR_RUNNER
                    //           }
                    //               IPC_AVANZAMENTO:
                    //                   IF Disp[IPC_MOTORE].stato<>LAVORO THEN
                    //                       OK_Condizione_Move_Dispositivo:=FALSE;
                    //                       set_trace(Code:=TRC_SAFETY_JOG_DEVICES, Asse:=IPC_MOTORE);
                    //                   END_IF;
                    //               IPC_LIGHT:
                    //                   IF cfg._4RUNNER_Mo1613=TRUE THEN
                    //                       IF Disp[IPC_MOTORE].stato<>LAVORO THEN
                    //                           OK_Condizione_Move_Dispositivo:=FALSE;
                    //                           set_trace(Code:=TRC_SAFETY_JOG_DEVICES, Asse:=IPC_MOTORE);
                    //                       END_IF;
                    //                   END_IF;
                    //           {
                    //           #endif  //Fine FOUR_RUNNER
                    //           }
                    //           {
                    //           #ifdef TAVOLI_SERPENTINE
                    //           }
                    //               TAVOLO_POST_ORIZZONTALE, TAVOLO_POST_ORIZZ_DX, TAVOLO_POST_ORIZZ_SX, TAVOLO_POST_ROTAZIONE:
                    //                   //Consentiti movimenti di chiusura tavoli verso la macchina solo con Z1 a 0° o 180°
                    //                   IF Stato=RIPOSO THEN
                    //                       IF ABS(Assi[Z1].PosAx.positioningState.actualPosition-0)>pm[Z1].ma_standstill_pos_tol AND
                    //                            ABS(Assi[Z1].PosAx.positioningState.actualPosition-180)>pm[Z1].ma_standstill_pos_tol THEN
                    //                           OK_Condizione_Move_Dispositivo:=FALSE;
                    //                           set_trace(Code:=TRC_SAFETY_JOG_DEVICES, Asse:=Z1);
                    //                       END_IF;
                    //                   END_IF;
                    //               TAVOLO_ANT_ORIZZONTALE:
                    //                   IF Stato=RIPOSO THEN
                    //                       //Consentiti movimenti di chiusura tavolo verso la macchina solo con Z1 a 0° o 180°
                    //                       IF ABS(Assi[Z1].PosAx.positioningState.actualPosition-0)>pm[Z1].ma_standstill_pos_tol AND
                    //                            ABS(Assi[Z1].PosAx.positioningState.actualPosition-180)>pm[Z1].ma_standstill_pos_tol THEN
                    //                           OK_Condizione_Move_Dispositivo:=FALSE;
                    //                           set_trace(Code:=TRC_SAFETY_JOG_DEVICES, Asse:=Z1);
                    //                       END_IF;
                    //                   END_IF;
                    //                   IF Stato=LAVORO THEN
                    //                       //Richiesta apertura tavolo orizzontale
                    //                       IF ReadDigitalInput(NumInput:=INP_TAVOLO_ANTERIORE_ALTO, Verifica:=TRUE)=FALSE THEN
                    //                           //Tavolo non è alto
                    //                           IF RunnerDXSX()=TRUE THEN
                    //                               IF Assi[Y1].PosAx.positioningState.actualPosition>1 AND Assi[Z1].PosAx.positioningState.actualPosition<179 THEN
                    //                                   //Con DXSX in processo non si può muovere se l^asse Y1 non è a 0° o 180°
                    //                                   OK_Condizione_Move_Dispositivo:=FALSE;
                    //                                   set_trace(Code:=TRC_SAFETY_JOG_DEVICES, Asse:=Y1);
                    //                               END_IF;
                    //                           ELSE
                    //                               IF Assi[Y1].PosAx.positioningState.actualPosition>1 THEN
                    //                                   //Non si può muovere se l^asse Y1 non è a 0°
                    //                                   OK_Condizione_Move_Dispositivo:=FALSE;
                    //                                   set_trace(Code:=TRC_SAFETY_JOG_DEVICES, Asse:=Y1);
                    //                               END_IF;
                    //                           END_IF;
                    //                       END_IF;
                    //                   END_IF;
                    //               TAVOLO_ANT_ROTAZIONE:
                    //                   //Consentiti movimenti di chiusura tavoli verso la macchina solo con Z1 a 0° o 180°
                    //                   IF Stato=RIPOSO THEN
                    //                       IF ABS(Assi[Z1].PosAx.positioningState.actualPosition-0)>pm[Z1].ma_standstill_pos_tol AND
                    //                            ABS(Assi[Z1].PosAx.positioningState.actualPosition-180)>pm[Z1].ma_standstill_pos_tol THEN
                    //                           OK_Condizione_Move_Dispositivo:=FALSE;
                    //                           set_trace(Code:=TRC_SAFETY_JOG_DEVICES, Asse:=Z1);
                    //                       END_IF;
                    //                   END_IF;
                    //                   IF ReadDigitalInput(NumInput:=INP_TAVOLO_ANTERIORE_FUORI_INGOMBRO, Verifica:=TRUE)=TRUE THEN
                    //                       //Tavolo anteriore orizzontale aperto
                    //                       IF RunnerDXSX()=TRUE THEN
                    //                           IF Assi[Y1].PosAx.positioningState.actualPosition>1 AND Assi[Z1].PosAx.positioningState.actualPosition<179 THEN
                    //                               //Con DXSX in processo non si può muovere se l^asse Y1 non è a 0° o 180°
                    //                               OK_Condizione_Move_Dispositivo:=FALSE;
                    //                               set_trace(Code:=TRC_SAFETY_JOG_DEVICES, Asse:=Y1);
                    //                           END_IF;
                    //                       ELSE
                    //                           IF Assi[Y1].PosAx.positioningState.actualPosition>1 THEN
                    //                               //Non si può muovere se l^asse Y1 non è a 0°
                    //                               OK_Condizione_Move_Dispositivo:=FALSE;
                    //                               set_trace(Code:=TRC_SAFETY_JOG_DEVICES, Asse:=Y1);
                    //                           END_IF;
                    //                   END_IF;
                    //               END_IF;
                    //           {
                    //           #endif  //Fine TAVOLI_SERPENTINE
                    //           }
                    //       {
                    //       #else	//Fine RUNNER
                    //       }
                              //Inizio macchine NO RUNNER
                              PALETTA:
                                  PosAx:= AsSynchronousAxisRef(Axes[Z1].PosAx);
                                  IF ABS(PosAx^.actualPosition)>pm[Z1].ma_tolerance AND Stato=DEVICES_STATUS#RIPOSO THEN
                                      OK_Condizione_Move_Dispositivo:=FALSE;
                                  END_IF;
                              SUPPORT_TIRANT:
                                  PosAx:= AsSynchronousAxisRef(Axes[X1].PosAx);
                                  IF PosAx^.actualPosition<=MAX(i_sys_MAX_X_SOSTEGNO_ALTO, cfg.QuotaAbbassoSostegnoTirante) THEN
                                      OK_Condizione_Move_Dispositivo:=FALSE;
                                      set_trace(Code:=TRC_SAFETY_JOG_DEVICES, Axis:=X1);
                                  END_IF;
                              CLAMP:
                                  IF ImpostaDiametroPinza(DiametroRichiesto:=programmi[PROGRAM_JOG].PinzaDiamMinMax)=FALSE THEN
                                      OK_Condizione_Move_Dispositivo:=FALSE;
                                      set_trace(Code:=TRC_SAFETY_JOG_DEVICES, Axis:=CLAMP);
                                  END_IF;
                                //   {
                                //   #ifdef SMART_SMART_A
                                //   }
                                //       {
                                //       #ifdef SMART
                                //       }
                                //           {
                                //           #ifndef BASCULANTE_ELETTRICO
                                //           }
                                //               BASCULANTE:
                                //                   IF i_sys_monitoring=1 AND ABS(Disp[BASCULANTE].limite2_lavoro-Disp[BASCULANTE].limite2_riposo)<0.1 THEN
                                //                       //Limiti calcolati da VGP sono uguali significa collisione e non si può movimentare il dispositivo
                                //                       OK_Condizione_Move_Dispositivo:=FALSE;
                                //                       set_trace(Code:=TRC_SAFETY_JOG_DEVICES, Asse:=BASCULANTE);
                                //                   ELSE
                                //                       IF Assi[V1].PosAx.positioningState.actualPosition-cfg.i_sys_postestabassaxmin>pm[V1].ma_standstill_pos_tol THEN
                                //                           iret:=Push_error(Code:=ERR_TESTA_NO_BASSA);
                                //                           OK_Condizione_Move_Dispositivo:=FALSE;
                                //                       END_IF;
                                //                   END_IF;
                                //           {
                                //           #endif  //Fine NO BASCULANTE_ELETTRICO
                                //           }
                                //       {
                                //       #endif  //Fine SMART
                                //       }
                                //       LOCKING_DXSX:
                                //           IF i_sys_monitoring=1 AND ABS(Disp[LOCKING_DXSX].limite2_lavoro-Disp[LOCKING_DXSX].limite2_riposo)<0.1 THEN
                                //               //Limiti calcolati da VGP sono uguali significa collisione e non si può movimentare il dispositivo
                                //               OK_Condizione_Move_Dispositivo:=FALSE;
                                //               set_trace(Code:=TRC_SAFETY_JOG_DEVICES, Asse:=LOCKING_DXSX);
                                //           ELSE
                                //               {
                                //               #ifdef SMART
                                //               }
                                //                   IF cfg.tiposlittamobile=TIPO_SLITTA_ELETTRICA THEN
                                //                       IF Clk_plus AND (Assi[W4].PosAx.positioningState.actualPosition>0) THEN
                                //                           //Richiesto tassello a SX, non si può fare con braccio minore di 45°
                                //                           IF Assi[Y1].PosAx.positioningState.actualPosition<45 THEN
                                //                               iret:=Push_error(Code:=ERR_SCOMPARSA_SLITTA);
                                //                               OK_Condizione_Move_Dispositivo:=FALSE;
                                //                           END_IF;
                                //                       ELSE
                                //                           IF Clk_minus AND (Assi[W4].PosAx.positioningState.actualPosition<0) THEN
                                //                               //Richiesto tassello a DX, non si può fare con braccio di curvatura supeiore a 145°
                                //                               IF Assi[Y1].PosAx.positioningState.actualPosition>POSY_SCOMPBLOCC_SX THEN
                                //                                   iret:=Push_error(Code:=ERR_SCOMPARSA_SLITTA);
                                //                                   OK_Condizione_Move_Dispositivo:=FALSE;
                                //                               END_IF;
                                //                           END_IF;
                                //                       END_IF;
                                //                   ELSE
                                //                       IF Disp[DISAPPEARANCE_ROLLERS].enable=TRUE THEN
                                //                           IF Disp[DISAPPEARANCE_ROLLERS].stato<>LAVORO THEN
                                //                               //Rulli non in posizione di scomparsa, il movimento del tassello morsa DX/SX è
                                //                               //condizionato dalla posizione del braccio di curvatura e dal tasto premuto
                                //                               IF Clk_plus AND (Assi[W4].PosAx.positioningState.actualPosition>0) THEN
                                //                                   //Richiesto tassello a SX, non si può fare con braccio minore di 45°
                                //                                   IF Assi[Y1].PosAx.positioningState.actualPosition<45 THEN
                                //                                       iret:=Push_error(Code:=ERR_SCOMPARSA_SLITTA);
                                //                                       OK_Condizione_Move_Dispositivo:=FALSE;
                                //                                   END_IF;
                                //                               ELSE
                                //                                   IF Clk_minus AND (Assi[W4].PosAx.positioningState.actualPosition<0) THEN
                                //                                       //Richiesto tassello a DX, non si può fare con braccio di curvatura supeiore a 145°
                                //                                       IF Assi[Y1].PosAx.positioningState.actualPosition>POSY_SCOMPBLOCC_SX THEN
                                //                                           iret:=Push_error(Code:=ERR_SCOMPARSA_SLITTA);
                                //                                           OK_Condizione_Move_Dispositivo:=FALSE;
                                //                                       END_IF;
                                //                                   END_IF;
                                //                               END_IF;
                                //                           END_IF;
                                //                       END_IF;
                                //                   END_IF;
                                //               {
                                //               #endif	//Fine SMART
                                //               }
                                //               {
                                //               #ifdef SMART_A
                                //               }
                                //                   IF Assi[U4].PosAx.positioningState.actualPosition>U4_Scomparsa+0.2 THEN
                                //                       //Rulli non in posizione di scomparsa, il movimento del tassello morsa DX/SX è
                                //                       //condizionato dalla posizione del braccio di curvatura e dal tasto premuto
                                //                       IF Clk_plus AND (Assi[W4].PosAx.positioningState.actualPosition>0) THEN
                                //                           //Richiesto tassello a SX, non si può fare con braccio minore di 45°
                                //                           IF Assi[Y1].PosAx.positioningState.actualPosition<45 THEN
                                //                               iret:=Push_error(Code:=ERR_SCOMPARSA_SLITTA);
                                //                               OK_Condizione_Move_Dispositivo:=FALSE;
                                //                           END_IF;
                                //                       ELSE
                                //                           IF Clk_minus AND (Assi[W4].PosAx.positioningState.actualPosition<0) THEN
                                //                               //Richiesto tassello a DX, non si può fare con braccio di curvatura supeiore a 145°
                                //                               IF Assi[Y1].PosAx.positioningState.actualPosition>POSY_SCOMPBLOCC_SX THEN
                                //                                   iret:=Push_error(Code:=ERR_SCOMPARSA_SLITTA);
                                //                                   OK_Condizione_Move_Dispositivo:=FALSE;
                                //                               END_IF;
                                //                           END_IF;
                                //                       END_IF;
                                //                   END_IF;
                                //               {
                                //               #endif  //Fine SMART_A
                                //               }
                                        //   END_IF;
                                      DISAPPEARANCE_ROLLERS:
                                          IF i_sys_monitoring=1 AND ABS(Disp[DISAPPEARANCE_ROLLERS].limite2_lavoro-Disp[DISAPPEARANCE_ROLLERS].limite2_riposo)<0.1 THEN
                                              //Limiti calcolati da VGP sono uguali significa collisione e non si può movimentare il dispositivo
                                              OK_Condizione_Move_Dispositivo:=FALSE;
                                              set_trace(Code:=TRC_SAFETY_JOG_DEVICES, Axis:=DISAPPEARANCE_ROLLERS);
                                          ELSE
                                              IF (Clk_minus OR Clk_plus) AND Disp[DISAPPEARANCE_ROLLERS].enable=TRUE THEN
                                                    PosAx:= AsSynchronousAxisRef(Axes[W4].PosAx);
                                                  IF PosAx^.actualPosition > 0 THEN
                                                      //Rulli lato DX si possono portare in posizione di lavoro solo se l^asse è sul limite positivo
                                                      IF PosAx^.actualPosition < PosAx^.PositionLimits_SW.MinPosition-1 THEN
                                                          iret:=Push_error(Code:=ERR_APRIRE_SLITTA_SPALLAMENTO);
                                                          OK_Condizione_Move_Dispositivo:=FALSE;
                                                      END_IF;
                                                  ELSE
                                                      //Rulli lato SX si possono portare in posizione di lavoro solo se l^asse è sul limite negativo
                                                      IF PosAx^.actualPosition > PosAx^.PositionLimits_SW.MinPosition+1 THEN
                                                          iret:=Push_error(Code:=ERR_APRIRE_SLITTA_SPALLAMENTO);
                                                          OK_Condizione_Move_Dispositivo:=FALSE;
                                                      END_IF;
                                              END_IF;
                                              IF Disp[LOCKING_DXSX].enable=TRUE AND cfg.bloccoscomparsabloccaggio=-1 THEN
                                                PosAx:= AsSynchronousAxisRef(Axes[Y1].PosAx);
                                                  IF PosAx^.actualPosition<POSY_SCOMPBLOCC_DX THEN
                                                      IF Disp[LOCKING_DXSX].stato<>DEVICES_STATUS#RIPOSO THEN
                                                          //Richiesta rulli in posizione di lavoro non si può
                                                          //eseguire con posizione Y inferiore a 35° e tassello
                                                          //bloccaggio in posizione diversa da DX
                                                          iret:=Push_error(Code:=ERR_TASSELLO_BLOCCAGGIO_DXSX);
                                                          OK_Condizione_Move_Dispositivo:=FALSE;
                                                      END_IF;
                                                  ELSE
                                                      IF PosAx^.actualPosition>POSY_SCOMPBLOCC_SX THEN
                                                          IF Disp[LOCKING_DXSX].stato<>DEVICES_STATUS#LAVORO THEN
                                                              //Richiesta rulli in posizione di lavoro non si può
                                                              //eseguire con posizione Y superiore a 145° e tassello
                                                              //bloccaggio in posizione diversa da SX
                                                              iret:=Push_error(Code:=ERR_TASSELLO_BLOCCAGGIO_DXSX);
                                                              OK_Condizione_Move_Dispositivo:=FALSE;
                                                          END_IF;
                                                      END_IF;
                                                  END_IF;
                                              END_IF;
                                          END_IF;
                                      END_IF;
                                //   {
                                //   #endif  //Fine SMART_SMART_A
                                //   }
                                //   {
                                //   #ifdef ELECTL_SAFETY %%%%
                                //   }
                                //       UNITA_FORATURA:
                                //           IF ReadDigitalInput(NumInput:=INP_POMPA_AVVIATA_FORATURA, Verifica:=1) = FALSE OR
                                //                ReadDigitalInput(NumInput:=INP_LIVELLO_OLIO_FORATURA, Verifica:=1) = FALSE THEN
                                //               iret:=Push_Error(Code:=ERR_POMPA_NON_PRONTA);
                                //               OK_Condizione_Move_Dispositivo:=FALSE;
                                //           END_IF;
                                //       FORATURA_IDRAULICA:
                                //           IF ReadDigitalInput(NumInput:=INP_POMPA_AVVIATA_FORATURA, Verifica:=1) = FALSE OR
                                //                ReadDigitalInput(NumInput:=INP_LIVELLO_OLIO_FORATURA, Verifica:=1) = FALSE THEN
                                //               iret:=Push_Error(Code:=ERR_POMPA_NON_PRONTA);
                                //               OK_Condizione_Move_Dispositivo:=FALSE;
                                //           END_IF;
                                //   {
                                //   #endif FINE ELECTL_SAFETY
                                //   }
                        //           {
                        //           #ifdef ELECTMRL
                        //           }
                        //               {
                        //               #ifdef TAVOLI_ELETTRICI
                        //               }
                        //                   TAVOLO_PNEUMATICO:
                        //                       IF assi[Y1].PosAx.positioningState.actualPosition <= 90 THEN
                        //                           iret:=Push_error(Code:=ERR_BRACCIO_NON_OPPOSTO);
                        //                           Ok_condizione_move_dispositivo:=FALSE;
                        //                       END_IF;
                        //               {
                        //               #endif //FINE TAVOLI_ELETTRICI
                        //               }
                        //           {
                        //           #endif //FINE ELECTMRL
                        //           }
                        //   {
                        //   #endif  //Fine NO RUNNER
                        //   }
                  END_CASE;
        //       {
        //       #endif //FINE NO PLAUNO_LIGHT
        //       }
        //       ;
        //   {
        //   #endif  //Fine NO EFLEX_DH4010
        //   }
      END_IF;
  END_FUNCTION
